	Version history:
	Date        | Version   | Author        | Remark
	----------------------------------------------------------------------------------------
	24/05/2019  | 0.1       | S. Nikodem    | First release MHS TIA 15.1
	14/06/2019  | 0.2       | M. Kurc       | Replacement of instruction if for direct write into variable, temporary variables review
	14/06/2019  | 0.3       | M. Kurc       | Communication error corrected
	19/06/2019  | 0.4       | M. Kurc       | Deleting error word
	25/06/2019  | 0.6       | M. Kurc       | Change interface q_UDT_VFDStatistic to iq_UDT_VFDStatistic
	04/07/2019  | 0.7       | S. Nikodem    | Add auto-parametrization fuction
	18/07/2019  | 0.8       | M. Kurc       | Deleting functions (denormaliztion, normalization, rpm-mm/s, mm/s-rpm)
	24/07/2019  | 2.0       | L. Klar       | 2.0 MHS library release TIA 15.1
	14/08.2019  | 2.1       | K. Pokorski   | Profinet number and HWID reading logic added
	09/09/2019  | 2.2       | S. Nikodem    | Complete rebuild block
	17/09/2019  | 2.3       | S. Nikodem    | Add ramp start/stop
	30/09/2019  | 2.4       | K. Pokorski   | Changed region 1 contents to FC
	30/09/2019  | 2.5       | K. Pokorski   | Implemented new VFD status
	30/09/2019  | 2.6       | L. Klar       | Actual speed connected to a new interface UDT, UDT interface changed
	11/10/2019  | 2.7       | S. Nikodem    | Added Interlock, quick stop, default ramp start/stop time = 20s, running statistic
	30/10/2019  | 2.8       | K. Pokorski   | Acceleration and deceleration calculating fixed
	30/10/2019  | 2.9       | K. Pokorski   | Internal warning and error handling changed
	20/11/2019  | 2.10      | S. Nikodem    | Configuration error
	20/11/2019  | 3.0       | P.Majka       | 3.0 MHS library release TIA 15.1
	03/12/2019  | 3.1       | S. Nikodem    | Change of direction
	20/12/2019  | 3.2       | S. Deulkar    | Used configureation error bit to report to conveyor block
	28/01/2020  | 3.3       | S. Nikodem    | Configuration error if speed setpoint is too high
	06/02/2020  | 3.4       | S. Nikodem    | Configuration error - Simulation mode bypass PNDeviceFound
	02/01/2020  | 3.5       | F.Baten       | Changed "UDT_VFD_Status" to be without positioning status
	04/03/2020  | 3.6       | F.Baten       | Output speed scaling based on measured speed at fixed output value, removal of gearratio and wheelendperrimeter
	01/05/2020  | 3.7       | F.Baten       | Reverted 3.6 modification measured speed
	18/06/2020  | 3.8       | L.Klar        | ix_PowerOK splitted to 24vOK and 400vOK
	23/06/2020  | 3.9       | L.Klar        | VFD running change to cover deceleration ramp, at speed condition changed to have False in standstill
	08/07/2020  | 3.10      | S.Theocharis  | Change VFD acknowledge to extended pulse & send acknowledge even with PN Slave error
	09/07/2020  | 3.11      | S.Theocharis  | Updated PO UDT
	10/07/2020  | 3.12      | S.Theocharis  | Comment out the PNSlave error from the VfdAvailable and ErrorActive variables to allo run in a ring topology
	22/07/2020  | 3.13      | K.Pokorski    | Protection against negative actual speed (int overflow)
	14/09/2020  | 3.14      | S.Nikodem     | VFDRunningFeedback error
	03/11/2020  | 3.15      | K.Pokorski    | Profinet ports diagnostics added
	06/01/2022  | 3.16      | M.Roijen      | Update new FB_Commissioning block
	21/02/2023  | 4.0       | F.Baten       | 4.0 Release TIA 17.5
	    *)

	REGION 1 - Get Device Profinet information

	    "FC_GetDevicePN"(is_PNDeviceName := #iUDT_VfdConfig.VFDPNDeviceName,
	                     ix_SimulationModeActive := #ix_SimulationModeActive,
	                     iqUDT_PND := #sUDT_PNDevice);


	    "FC_GetPNPortStatus"(ii_NumberOfPorts := #ci_NumberOfProfinetPorts,
	                         iUDT_DevicePNInfo := #sUDT_PNDevice,
	                         qa_PortFault => #sa_PNPortsStatus);

	END_REGION

	REGION 2 - Reset errors

	    IF #iqUDT_ConveyorInterface.InternalErrorReset                           // Reser errors when Reset is given
	    THEN

	        #sUDT_Status.PNSlaveNotonline := FALSE;
	        #sUDT_Status.PNSlaveError := FALSE;
	        #sUDT_Status.InternalError := FALSE;
	        #sUDT_Status.VFDRunningFeedbackError := FALSE;
	        #sUDT_Status.PNSlaveWarning := FALSE;

	    END_IF;


	    // Create  extended pulse for VFD Reset
	    #sFB_TimerOnOffDelayVFDReset(iudi_OnDelayTime := 0,
	                                 iudi_OffDelayTime := 200,
	                                 ix_SignalToDelay := #iqUDT_ConveyorInterface.InternalErrorReset,
	                                 ix_Enable := TRUE);

	END_REGION

	REGION 3 - Hardware checks
	    // Hardware will only be available after the delay, so the device has time for the initialisation
	    #sFB_TimerOnOffDelayCheck24V(iudi_OnDelayTime := 2000,
	                                 ix_SignalToDelay := #ix_24vOk);

	    #sx_24vOk := #sFB_TimerOnOffDelayCheck24V.qx_DelayedSignal;

	    #sFB_TimerOnOffDelayCheck400V(iudi_OnDelayTime := 2000,
	                                  ix_SignalToDelay := #ix_400vOk);

	    #sx_400vOk := #sFB_TimerOnOffDelayCheck400V.qx_DelayedSignal;

	    // Check if PN device is online
	    IF NOT "DB_ProfinetDiagnostic".ProfinetNetworks[#sUDT_PNDevice.PNNetworknumber].DeviceStatus[#sUDT_PNDevice.PNDeviceNumber].DeviceState.Exist
	        AND NOT #ix_SimulationModeActive
	        AND #sx_24vOk
	    THEN
	        #sUDT_Status.PNSlaveNotonline := TRUE;

	    END_IF;

	    // Check if PN ports are healthy
	    IF #sa_PNPortsStatus[1] XOR #sa_PNPortsStatus[2] THEN
	        #sUDT_Status.PNSlaveWarning := TRUE;
	    END_IF;


	    // Check if PN device has an error
	    IF "DB_ProfinetDiagnostic".ProfinetNetworks[#sUDT_PNDevice.PNNetworknumber].DeviceStatus[#sUDT_PNDevice.PNDeviceNumber].DeviceState.Error
	        AND NOT #ix_SimulationModeActive
	        AND #sx_24vOk
	        AND NOT #sUDT_Status.PNSlaveWarning
	    THEN
	        #sUDT_Status.PNSlaveError := TRUE;
	    END_IF;

	    // Set bit when PN device is healthy (online and no error)
	    #sx_PNDeviceHealthy := NOT #sUDT_Status.PNSlaveNotonline
	    AND NOT #sUDT_Status.PNSlaveError
	    AND #sUDT_PNDevice.PNDeviceFound
	    AND #sx_24vOk;

	    // Set hardware available bit when all conditions are met
	    #sx_HardwareAvailable := (#sx_24vOk
	    AND #sx_PNDeviceHealthy)
	    OR #ix_SimulationModeActive;


	    // VFD is ready for operation if hardware ok
	    #sx_VFD_Available := #sx_HardwareAvailable;

	END_REGION

	REGION 4 - Check errors and warnings

	    // Check if the VFD has a warning
	    #sUDT_Status.InternalWarning := #iUDT_VfdInputs.ZSW_1.AlarmActive;

	    // Copy warning code to status DB when warning active
	    IF #iUDT_VfdInputs.ZSW_1.AlarmActive
	    THEN

	        #sUDT_Status.ErrorCode := UINT_TO_INT(#iUDT_VfdInputs.AlarmCode);

	    END_IF;

	    // Check if the VFD has an error
	    #sUDT_Status.InternalError := #iUDT_VfdInputs.ZSW_1.FaultActive AND NOT #sx_StartMeasuring;

	    // Copy error code to status DB when error active
	    IF #iUDT_VfdInputs.ZSW_1.FaultActive
	    THEN

	        #sUDT_Status.ErrorCode := UINT_TO_INT(#iUDT_VfdInputs.FaultCode);

	    END_IF;

	    // Reset error code if warning and error not available
	    IF (NOT #iUDT_VfdInputs.ZSW_1.AlarmActive
	        AND NOT #iUDT_VfdInputs.ZSW_1.FaultActive)
	    THEN

	        #sUDT_Status.ErrorCode := 0;

	    END_IF;

	END_REGION

	REGION 5 - Check if configuration is ok for commissioning purposes

	    IF #iUDT_VfdConfig.WheelEndPerimeter > 0.0                                         // If perimeter of wheel at the end of gear is greater than 0
	        AND #iUDT_VfdConfig.GearRatio > 0.0                                            // and gear ratio is greater than 0
	        AND #iUDT_VfdConfig.ReferenceRPM > 0.0                                             // and maximum speed is greater than 0
	        AND #iUDT_VfdConfig.VFDRampUpTime > 0                                          // and ramp up time is greater than 0
	        AND #iUDT_VfdConfig.VFDRampDownTime > 0                                        // and ramp down time is greater than zero
	        AND #iUDT_VfdConfig.VFDStartupTime > 0.0                                       // and startup time is greater then zero
	        AND 2 * #cudi_DefaultRampUpTime > #iUDT_VfdConfig.VFDRampUpTime                // and ramp up time is not greater two time than default ramp up time
	        AND 2 * #cudi_DefaultRampDownTime > #iUDT_VfdConfig.VFDRampDownTime            // and ramp down time is not greater two time than default ramp down time

	        AND (#sUDT_PNDevice.PNDeviceFound                                              // and device not found in PN structure
	        OR #ix_SimulationModeActive)                                                    // or simulation mode is active
	    THEN
	        #sx_ConfigurationError := FALSE;                                                // Reset configuration error
	    ELSE
	        #sx_ConfigurationError := TRUE;                                                 // Set configuration error
	    END_IF;

	END_REGION

	REGION 6 - Speed handling

	    // Calculate actual speed in mm/s
	    #si_ActualSpeed := REAL_TO_INT((((INT_TO_REAL(#iUDT_VfdInputs.ActualSpeed) / #cr_MaximumOutput) * #iUDT_VfdConfig.ReferenceRPM) / #iUDT_VfdConfig.GearRatio) * #iUDT_VfdConfig.WheelEndPerimeter / 60.0);

	    // Reversal actual speed
	    IF #iUDT_VfdConfig.DirectionReversal THEN

	        #si_ActualSpeed := #si_ActualSpeed * -1;

	    END_IF;

	    // Calculate actual speed setpoint
	    #sr_ActualSpeedSetpoint := ((DINT_TO_REAL(INT_TO_DINT(#iqUDT_ConveyorInterface.SpeedSetpoint) * 60) / #iUDT_VfdConfig.WheelEndPerimeter) * #iUDT_VfdConfig.GearRatio);

	    // Check if speed setpoint is reached
	    #sx_SpeedSetpointReached := (ABS(#si_ActualSpeed) >= (#iqUDT_ConveyorInterface.SpeedSetpoint - #iUDT_VfdConfig.SpeedSetpointWindow))
	    AND (ABS(#si_ActualSpeed) <= (#iqUDT_ConveyorInterface.SpeedSetpoint + #iUDT_VfdConfig.SpeedSetpointWindow));
	END_REGION

	REGION 7 - Prepare output data VFD
	    REGION 7.1 - Set speed setpoint in forward and reverse directory

	        // If motor stopped and Run forward is requested and interlock forward is active, the speed setpoint is loaded to run forward.
	        IF (#iUDT_VfdInputs.ActualSpeed = 0) AND #iqUDT_ConveyorInterface.RunFwd AND #iUDT_VfdConfig.InterlockFwd
	        THEN
	            #sx_RunVFDForward := TRUE;
	            #sx_RunVFDReverse := FALSE;
	        END_IF;

	        // If motor stopped and Run reverse is requested and interlock reverse is active, the speed setpoint is loaded to run reverse.
	        IF (#iUDT_VfdInputs.ActualSpeed = 0) AND #iqUDT_ConveyorInterface.RunRvs AND #iUDT_VfdConfig.InterlockRvs
	        THEN
	            #sx_RunVFDReverse := TRUE;
	            #sx_RunVFDForward := FALSE;
	        END_IF;

	    END_REGION

	    REGION 7.2 - Stopping

	        // Create trigger when direction signal falling
	        #sF_TRIG_RunFwd(CLK := #iqUDT_ConveyorInterface.RunFwd);
	        #sF_TRIG_RunRvs(CLK := #iqUDT_ConveyorInterface.RunRvs);

	        // When no run signal is given the VFD should stop
	        IF NOT #iqUDT_ConveyorInterface.RunRvs AND NOT #iqUDT_ConveyorInterface.RunFwd
	            OR (#iqUDT_ConveyorInterface.RunRvs AND #iqUDT_ConveyorInterface.RunFwd)
	            OR #sF_TRIG_RunRvs.Q
	            OR #sF_TRIG_RunFwd.Q

	        THEN
	            #sx_RunVFDReverse := FALSE;
	            #sx_RunVFDForward := FALSE;
	        END_IF;

	        IF NOT #sx_RunVFDReverse AND NOT #sx_RunVFDForward AND (#iUDT_VfdInputs.ActualSpeed <> 0)
	        THEN
	            #sx_VFDStopping := TRUE;
	        ELSE
	            #sx_VFDStopping := FALSE;
	        END_IF;

	    END_REGION

	    REGION 7.3 - Check for enable operation signal

	        #sx_EnableOperation := #sx_VFD_Available AND #sx_400vOk AND NOT #sx_ConfigurationError AND (#sx_RunVFDForward OR #sx_RunVFDReverse); // add communication error

	    END_REGION

	    REGION 7.4 - Write acceleration and deceleration value to drive
	        // Write accceleration value to VFD
	        #qUDT_VfdOutputs.SetpointAcceleration := REAL_TO_INT(#cr_MaximumOutput / UDINT_TO_REAL(#cudi_DefaultRampUpTime) * UDINT_TO_REAL(#iUDT_VfdConfig.VFDRampUpTime));        //Recalculating Acceleration ramp

	        // Write deceleration value to VFD
	        #qUDT_VfdOutputs.SetpointDeceleration := REAL_TO_INT(#cr_MaximumOutput / UDINT_TO_REAL(#cudi_DefaultRampDownTime) * UDINT_TO_REAL(#iUDT_VfdConfig.VFDRampDownTime));      //Recalculating Deceleration ramp

	    END_REGION

	END_REGION

	REGION 8 - Auto Commisioning

	    REGION 8.1 Extract telegram's HW_ID

	        IF (#ix_StartCommissioning)
	        THEN

	            #si_Log2GeoReturn := LOG2GEO(LADDR := "DB_ProfinetDiagnostic".ProfinetNetworks[#sUDT_PNDevice.PNNetworknumber].DeviceStatus[#sUDT_PNDevice.PNDeviceNumber].DeviceState.HW_ID, GEOADDR := #sv_VFDGeoStruct);       // "LOG2GEO" to get profinet network number
	            #sv_VFDGeoStruct.AREA := #ci_VFDArea;                                                                                                                                                                               // Set IO Profinet devices area ID
	            #sv_VFDGeoStruct.HWTYPE := #ci_SubmoduleHWType;                                                                                                                                                                     // Set submodule HW_type number
	            #sv_VFDGeoStruct.STATION := INT_TO_UINT(#sUDT_PNDevice.PNDeviceNumber);                                                                                                                                            // Set device's profinet number
	            #sv_VFDGeoStruct.SLOT := #ci_TelegramSlot;                                                                                                                                                                          // Set free telegram slot
	            #sv_VFDGeoStruct.SUBSLOT := #ci_TelegramSubslot;                                                                                                                                                                    // Set free telegram subslot

	            #si_Geo2LogReturn := GEO2LOG(GEOADDR := #sv_VFDGeoStruct, LADDR => #shw_VFD_Telegram);                                                                                                                              // "GEO2LOG" to get free telegram's HW_ID

	        END_IF;

	    END_REGION

	    REGION 8.2 Run auto - commissioning

	        // Using commissioning block to write/read parameter. Start parametrization if rise edge trigger from start commissionig signal
	        #sFB_Commissioning(ix_Enable := #ix_StartCommissioning,
	                           ihw_SinaParamHardwareId := #shw_VFD_Telegram,                    // Set hardware id ,
	                           iUDT_MotorConfig := #iUDT_MotorData,
	                           qx_StartMeasuring => #sx_StartMeasuring,                         // Set start measuring signal
	                           iqx_GoToNextStep := #iqx_GoToNextStepCommissioning);             // Set/Reset signal go to next step


	    END_REGION ;

	END_REGION

	REGION 9 - Write outputs to VFD

	    REGION 9.1 - Write control word 1


	        #qUDT_VfdOutputs.STW_1.ControlViaPLC := TRUE;
	        #qUDT_VfdOutputs.STW_1.DirectionReversal := FALSE;
	        #qUDT_VfdOutputs.STW_1.ONOFF1 := #sx_EnableOperation OR #sx_StartMeasuring;
	        #qUDT_VfdOutputs.STW_1.OFF2 := TRUE;
	        #qUDT_VfdOutputs.STW_1.OFF3 := #ix_QuickStopDisable;
	        #qUDT_VfdOutputs.STW_1.EnableOperation := #sx_RunVFDReverse OR #sx_RunVFDForward OR #iUDT_VfdInputs.ActualSpeed <> 0 OR #sx_StartMeasuring;
	        #qUDT_VfdOutputs.STW_1.DoNotDisableRFG := TRUE;
	        #qUDT_VfdOutputs.STW_1.EnableRFG := TRUE;
	        #qUDT_VfdOutputs.STW_1.EnableSetpoint := TRUE;
	        #qUDT_VfdOutputs.STW_1.Acknowledge := #sFB_TimerOnOffDelayVFDReset.qx_DelayedSignal;


	        IF (NOT #sx_VFD_Available OR NOT #sx_400vOk) AND NOT #sx_StartMeasuring
	        THEN

	            #qUDT_VfdOutputs.STW_1.ForceDormantErrorTest := FALSE;
	            #qUDT_VfdOutputs.STW_1.SpareBit9 := FALSE;
	            #qUDT_VfdOutputs.STW_1.DirectionReversal := FALSE;
	            #qUDT_VfdOutputs.STW_1.SpareBit12 := FALSE;
	            #qUDT_VfdOutputs.STW_1.SpareBit13 := FALSE;
	            #qUDT_VfdOutputs.STW_1.SpareBit14 := FALSE;
	            #qUDT_VfdOutputs.STW_1.SpareBit15 := FALSE;
	            #qUDT_VfdOutputs.STW_1.ONOFF1 := FALSE;
	            #qUDT_VfdOutputs.STW_1.OFF2 := FALSE;
	            #qUDT_VfdOutputs.STW_1.OFF3 := FALSE;
	            #qUDT_VfdOutputs.STW_1.EnableOperation := FALSE;
	            #qUDT_VfdOutputs.STW_1.DoNotDisableRFG := FALSE;
	            #qUDT_VfdOutputs.STW_1.EnableRFG := FALSE;
	            #qUDT_VfdOutputs.STW_1.EnableSetpoint := FALSE;
	            #qUDT_VfdOutputs.SpeedSetpoint := 0;

	        END_IF;

	    END_REGION

	    REGION 9.2 - Write speed setpoint to drive

	        // Calculate normalized speed setpoint
	        #qUDT_VfdOutputs.SpeedSetpoint := REAL_TO_INT((#sr_ActualSpeedSetpoint / #iUDT_VfdConfig.ReferenceRPM) * #cr_MaximumOutput);
	        IF #qUDT_VfdOutputs.SpeedSetpoint > #cr_MaximumOutput
	        THEN
	            #qUDT_VfdOutputs.SpeedSetpoint := REAL_TO_INT(#cr_MaximumOutput);
	        END_IF;

	        // The conveyor stopped and may now run in reverse direction
	        IF (#sx_RunVFDReverse AND NOT #iUDT_VfdConfig.DirectionReversal)
	            OR (#sx_RunVFDForward AND #iUDT_VfdConfig.DirectionReversal)
	        THEN
	            #qUDT_VfdOutputs.SpeedSetpoint := #qUDT_VfdOutputs.SpeedSetpoint * -1;
	        END_IF;

	        // Clear speed setpoint when no run request or above direction request or is configuration error
	        IF (NOT #sx_RunVFDForward AND NOT #sx_RunVFDReverse)
	            OR #sx_ConfigurationError
	        THEN
	            #qUDT_VfdOutputs.SpeedSetpoint := 0;
	        END_IF;

	    END_REGION

	END_REGION

	REGION 10 - Check if motor is running

	    //The moto should start running after specific time. If not the VFDRunningFeedback error occured
	    #sFB_TimerOnOffDelayVFDRunningFeedbackError(iudi_OnDelayTime := #iUDT_VfdConfig.VFDStartupTime,
	                                                ix_SignalToDelay := #sx_EnableOperation AND NOT (#si_ActualSpeed <> 0));

	    IF #sFB_TimerOnOffDelayVFDRunningFeedbackError.qx_DelayedSignal THEN

	        #sUDT_Status.VFDRunningFeedbackError := TRUE;

	    END_IF;

	END_REGION

	REGION 11 - Copy signals to interface DB and to status output UDT
	    // Create internal error status
	    #sx_ErrorActive := #sUDT_Status.PNSlaveNotonline
	    OR #sUDT_Status.VFDRunningFeedbackError
	    //  OR #s_UDT_Status.PNSlaveError Commented out by AST to allow run in ring topology v3.12
	    OR #sUDT_Status.InternalError;

	    // Write interface bits
	    #iqUDT_ConveyorInterface.VFDRunning := #iUDT_VfdInputs.ZSW_1.Ready AND #sx_VFD_Available AND (#iqUDT_ConveyorInterface.ActualSpeed <> 0 OR #iUDT_VfdInputs.ZSW_1.OperationEnabled);   // Write true on output Conveyor interface structure if VFD is in operation and motor is turning
	    #iqUDT_ConveyorInterface.VFDatSpeed := #sx_SpeedSetpointReached AND #sx_VFD_Available AND #si_ActualSpeed <> 0;                                                                                                  // Copy setpoint speed reached state from static to the output conveyor interface structure
	    #iqUDT_ConveyorInterface.InternalWarningVFD := #iUDT_VfdInputs.ZSW_1.AlarmActive;                                                                                                      // Set the internal VFD warning bit if any warning is active
	    #iqUDT_ConveyorInterface.InternalErrorVFD := #sx_ErrorActive;                                                                                                                           // Set the internal VFD error bit if any fault is active
	    #iqUDT_ConveyorInterface.ActualSpeed := #si_ActualSpeed;                                                                                                                                // Copy the calculated value to the output
	    #iqUDT_ConveyorInterface.ConfigurationError := #iqUDT_ConveyorInterface.ConfigurationError OR #sx_ConfigurationError;

	    // Copy error status to output
	    #qUDT_HMIStatus := #sUDT_Status;

	END_REGION

	REGION 12 - Statistic
	    // Create trigger on error and create statistics for profinet slave not online
	    #sR_TRIG_PNSlaveNotOnline(CLK := #sUDT_Status.PNSlaveNotonline);                                        // Detect the rising edge of the error

	    IF #iqUDT_ConveyorInterface.ResetStatistics OR #sUDT_Status.PNSlaveNotonline
	    THEN

	        "FC_Statistics"(ix_Reset := #iqUDT_ConveyorInterface.ResetStatistics,
	                        ix_Activate := #sUDT_Status.PNSlaveNotonline,
	                        ix_RTrigActivate := #sR_TRIG_PNSlaveNotOnline.Q,
	                        iqUDT_Statistics := #iqUDT_VfdStatistics.PNSlaveNotOnline);
	    END_IF;

	    // Create trigger on error and create statistics for profinet slave error
	    #sR_TRIG_PNSlaveError(CLK := #sUDT_Status.PNSlaveError);                                        // Detect the rising edge of the error

	    IF #iqUDT_ConveyorInterface.ResetStatistics OR #sUDT_Status.PNSlaveError
	    THEN

	        "FC_Statistics"(ix_Reset := #iqUDT_ConveyorInterface.ResetStatistics,
	                        ix_Activate := #sUDT_Status.PNSlaveError,
	                        ix_RTrigActivate := #sR_TRIG_PNSlaveError.Q,
	                        iqUDT_Statistics := #iqUDT_VfdStatistics.PNSlaveError);
	    END_IF;

	    // Create trigger on error and create statistics for internal VFD Error
	    #sR_TRIG_VFDInternalError(CLK := #sUDT_Status.InternalError);                                        // Detect the rising edge of the error

	    IF #iqUDT_ConveyorInterface.ResetStatistics OR #sUDT_Status.InternalError
	    THEN

	        "FC_Statistics"(ix_Reset := #iqUDT_ConveyorInterface.ResetStatistics,
	                        ix_Activate := #sUDT_Status.InternalError,
	                        ix_RTrigActivate := #sR_TRIG_VFDInternalError.Q,
	                        iqUDT_Statistics := #iqUDT_VfdStatistics.VFDInternalError);
	    END_IF;

	    // Create trigger on running signal and create statistics for running status
	    #sR_TRIG_Running(CLK := #iqUDT_ConveyorInterface.VFDRunning);                                        // Detect the rising edge of the signal

	    IF #iqUDT_ConveyorInterface.ResetStatistics OR #iqUDT_ConveyorInterface.VFDRunning
	    THEN

	        "FC_Statistics"(ix_Reset := #iqUDT_ConveyorInterface.ResetStatistics,
	                        ix_Activate := #iqUDT_ConveyorInterface.VFDRunning,
	                        ix_RTrigActivate := #sR_TRIG_Running.Q,
	                        iqUDT_Statistics := #iqUDT_VfdStatistics.Running);
	    END_IF;

	END_REGION
END_FUNCTION_BLOCK

FUNCTION_BLOCK "FB_Unloader"
TITLE = FB_Unloader
{ S7_Optimized_Access := 'TRUE' }
AUTHOR : MHSE
FAMILY : Equimpent
VERSION : 3.0
// ATTRIBUTES
// AUTO_NUMBER = True
// BLOCK_NUMBER = 232
// END_ATTRIBUTES
//Function block to control unloader.
   VAR_INPUT
      iUDT_UnloaderConfiguration { ExternalAccessible := 'False'; ExternalVisible := 'False'; ExternalWritable := 'False'} : "UDT_UnloaderConfiguration";   //   Unloader configuration structure
      ix_SafetyReset { ExternalAccessible := 'False'; ExternalVisible := 'False'; ExternalWritable := 'False'} : Bool;   //  Safety reset
      ix_SafetyOk { ExternalAccessible := 'False'; ExternalVisible := 'False'; ExternalWritable := 'False'} : Bool;   //   TRUE when Safety Circuit of the Conveyor is healthy
      ix_24vOk { ExternalAccessible := 'False'; ExternalVisible := 'False'; ExternalWritable := 'False'} : Bool;   //   TRUE when 24VDC is healthy
      ix_400vOk { ExternalAccessible := 'False'; ExternalVisible := 'False'; ExternalWritable := 'False'} : Bool;   //   TRUE when 400VAC is healthy
      ix_ProfinetOk { ExternalAccessible := 'False'; ExternalVisible := 'False'; ExternalWritable := 'False'} : Bool;   //   TRUE when the PN node(s) of VSU are OK
      ix_ReadyUnload { ExternalAccessible := 'False'; ExternalVisible := 'False'; ExternalWritable := 'False'} : Bool;   //   TRUE when Unloader is ready to unload
      ix_Running { ExternalAccessible := 'False'; ExternalVisible := 'False'; ExternalWritable := 'False'} : Bool;   //   TRUE when Unloader is running
      ix_TooLongParcel { ExternalAccessible := 'False'; ExternalVisible := 'False'; ExternalWritable := 'False'} : Bool;   //   TRUE when Unloader has detected a too long parcel (stopped)
      ix_VFDError { ExternalAccessible := 'False'; ExternalVisible := 'False'; ExternalWritable := 'False'} : Bool;   //   TRUE when Unloader has an VFD error
      ix_Healthy { ExternalAccessible := 'False'; ExternalVisible := 'False'; ExternalWritable := 'False'} : Bool;   //   TRUE when Unloader has no Errors
      ix_PECEoS { ExternalAccessible := 'False'; ExternalVisible := 'False'; ExternalWritable := 'False'} : Bool;   //   TRUE when the end of section photoeye is not blocked
      ix_ManualControlled { ExternalAccessible := 'False'; ExternalVisible := 'False'; ExternalWritable := 'False'} : Bool;   //   Unloader is controlled by
      ix_ExternalRequestDieBack { ExternalAccessible := 'False'; ExternalVisible := 'False'; ExternalWritable := 'False'} : Bool;   //   External request die back
      ix_ExternalRequestHold { ExternalAccessible := 'False'; ExternalVisible := 'False'; ExternalWritable := 'False'} : Bool;   //   External request hold
      ix_ResetEnergySave { ExternalAccessible := 'False'; ExternalVisible := 'False'; ExternalWritable := 'False'} : Bool;   //   Reset energy save mode timer
      ix_HardwareOk { ExternalAccessible := 'False'; ExternalVisible := 'False'; ExternalWritable := 'False'} : Bool;   //  TRUE when  hardware is Ok
   END_VAR

   VAR_OUTPUT
      qUDT_HMIStatus { ExternalAccessible := 'False'; ExternalVisible := 'False'; ExternalWritable := 'False'} : "UDT_UnloaderStatus";   //   HMI status structure
      qUDT_Status { ExternalAccessible := 'False'; ExternalVisible := 'False'; ExternalWritable := 'False'} : "UDT_CommonStatus";   //   Common status structure
      qi_SpeedSelect { ExternalAccessible := 'False'; ExternalVisible := 'False'; ExternalWritable := 'False'} : Int;   //   Speed select (slow, normal or fast)
      qx_ReleaseUnload { ExternalAccessible := 'False'; ExternalVisible := 'False'; ExternalWritable := 'False'} : Bool;   //   Release Unloader
      qx_EStopReset { ExternalAccessible := 'False'; ExternalVisible := 'False'; ExternalWritable := 'False'} : Bool;
      qx_FaultReset { ExternalAccessible := 'False'; ExternalVisible := 'False'; ExternalWritable := 'False'} : Bool;
   END_VAR

   VAR_IN_OUT
      iqUDT_EquipmentControl : "UDT_EquipmentControl";   //   Equipment control structure
      iqUDT_UnloaderCommand : "UDT_UnloaderCommand";   //   Unloader HMI control
      iqUDT_HandShake : "UDT_ConveyorHandshake";   //   Handshake structure
      iqUDT_EquipmentInterface : "UDT_ConveyorInterface";   //   Equipment interface structure
      iqUDT_Statistics : "UDT_UnloaderStatistics";   //   Statistics structure
   END_VAR

   VAR
      sUDT_CommonStatus { ExternalAccessible := 'False'; ExternalVisible := 'False'; ExternalWritable := 'False'; S7_SetPoint := 'False'} : "UDT_CommonStatus";   //   Common status structure
      sUDT_CommonStatusOld { ExternalAccessible := 'False'; ExternalVisible := 'False'; ExternalWritable := 'False'; S7_SetPoint := 'False'} : "UDT_CommonStatus";   //   Auxiliary status structure
      sUDT_HMIStatus { ExternalAccessible := 'False'; ExternalVisible := 'False'; ExternalWritable := 'False'; S7_SetPoint := 'False'} : "UDT_UnloaderStatus";   //   HMI status structure
      s_FB_TimerOnOffDelaySafetyOKPulse { ExternalAccessible := 'False'; ExternalVisible := 'False'; ExternalWritable := 'False'; S7_SetPoint := 'False'} : "FB_TimerOnOffDelay";
      sFB_PECEoSFiltered { ExternalAccessible := 'False'; ExternalVisible := 'False'; ExternalWritable := 'False'; S7_SetPoint := 'False'} : "FB_TimerOnOffDelay";   //   Filtering end of section photo eye signal
      sFB_PECEoSJamTimer { ExternalAccessible := 'False'; ExternalVisible := 'False'; ExternalWritable := 'False'; S7_SetPoint := 'False'} : "FB_TimerOnOffDelay";   //   Timer to detect photo eye jam
      sFB_EnergySaveTimer { ExternalAccessible := 'False'; ExternalVisible := 'False'; ExternalWritable := 'False'; S7_SetPoint := 'False'} : "FB_TimerOnOffDelay";   //   Timer to start energy save mode
      sFB_PEC { ExternalAccessible := 'False'; ExternalVisible := 'False'; ExternalWritable := 'False'; S7_SetPoint := 'False'} : "FB_PEC";   //   FB PEC block for PEC Jam status
      sR_TRIG_PEC_EoSFiltered {InstructionName := 'R_TRIG'; LibVersion := '1.0'; ExternalAccessible := 'False'; ExternalVisible := 'False'; ExternalWritable := 'False'; S7_SetPoint := 'False'} : R_TRIG;   //   Rising edge trigger end of section photo eye filtered
      sF_TRIG_PEC_EoSFiltered {InstructionName := 'F_TRIG'; LibVersion := '1.0'; ExternalAccessible := 'False'; ExternalVisible := 'False'; ExternalWritable := 'False'; S7_SetPoint := 'False'} : F_TRIG;   //   Falling edge trigger end of section photo eye filtered
      sR_TRIG_EnergySave {InstructionName := 'R_TRIG'; LibVersion := '1.0'; ExternalAccessible := 'False'; ExternalVisible := 'False'; ExternalWritable := 'False'; S7_SetPoint := 'False'} : R_TRIG;   //   Rising edge for energy save
      sR_TRIG_ConveyorUp {InstructionName := 'R_TRIG'; LibVersion := '1.0'; ExternalAccessible := 'False'; ExternalVisible := 'False'; ExternalWritable := 'False'; S7_SetPoint := 'False'} : R_TRIG;   //   Rising edge of automatic active
      sR_TRIG_ConveyorDown {InstructionName := 'R_TRIG'; LibVersion := '1.0'; ExternalAccessible := 'False'; ExternalVisible := 'False'; ExternalWritable := 'False'; S7_SetPoint := 'False'} : R_TRIG;   //   Rising edge of automatic not active
      sR_TRIG_VFDError {InstructionName := 'R_TRIG'; LibVersion := '1.0'; ExternalAccessible := 'False'; ExternalVisible := 'False'; ExternalWritable := 'False'; S7_SetPoint := 'False'} : R_TRIG;   //   Rising edge of VFD error
      sR_TRIG_NotHealthy {InstructionName := 'R_TRIG'; LibVersion := '1.0'; ExternalAccessible := 'False'; ExternalVisible := 'False'; ExternalWritable := 'False'; S7_SetPoint := 'False'} : R_TRIG;   //   Rising edge trigger if extendable not healthy
      sR_TRIG_TooLongParcel {InstructionName := 'R_TRIG'; LibVersion := '1.0'; ExternalAccessible := 'False'; ExternalVisible := 'False'; ExternalWritable := 'False'; S7_SetPoint := 'False'} : R_TRIG;   //   Rising edge trigger for too long parcel
      s_R_TRIG_SafetyOK {InstructionName := 'R_TRIG'; LibVersion := '1.0'; ExternalAccessible := 'False'; ExternalVisible := 'False'; ExternalWritable := 'False'; S7_SetPoint := 'False'} : R_TRIG;
      si_AuxEnergySave { ExternalAccessible := 'False'; ExternalVisible := 'False'; ExternalWritable := 'False'} : Int;   //   Auxiliery energy save
      sx_Disabled { ExternalAccessible := 'False'; ExternalVisible := 'False'; ExternalWritable := 'False'} : Bool;   //   Operation is enabled
      sx_Ready { ExternalAccessible := 'False'; ExternalVisible := 'False'; ExternalWritable := 'False'} : Bool;   //   Conveyor Ready to operate in Automatic mode
      sx_StartReceived { ExternalAccessible := 'False'; ExternalVisible := 'False'; ExternalWritable := 'False'} : Bool;   //   Start command received from system
      sx_PEC_EoSFiltered { ExternalAccessible := 'False'; ExternalVisible := 'False'; ExternalWritable := 'False'} : Bool;   //   End of section photo eye filtered
      sx_EnergySaveActive { ExternalAccessible := 'False'; ExternalVisible := 'False'; ExternalWritable := 'False'} : Bool;   //   Active energy save mode
      sx_AutomaticActive { ExternalAccessible := 'False'; ExternalVisible := 'False'; ExternalWritable := 'False'} : Bool;   //   Automatic active
   END_VAR


BEGIN
	(*
	----------------------------------------------------------------------------------------

	Version history:
	Date        | Version   | Author        | Remark
	----------------------------------------------------------------------------------------
	24/05/2019  | 0.1       | F.Baten       | first release MHS TIA 15.1
	17/06/2019  | 0.3       | L.Klar        | Manual mode added to "UDT_EquipmentControl"
	24/07/2019  | 2.0       | L.Klar        | 2.0 MHS library release TIA 15.1
	14/10/2019  | 2.1       | L.Klar        | Updated status structure
	15/10/2019  | 2.2       | S.Deulkar     | Deleted unused symbol, added statistcs, rearrange structure
	04/11/2019  | 2.3       | L.Klar        | First scan bit changed from memory bit to DB variable
	12/11/2019  | 3.0       | P.Majka       | 3.0 MHS library release TIA 15.1
	04/03/2020  | 3.1       | P.Majka       | Adapting reviews, repair statistics for too long parcels
	31/03/2020  | 3.2       | F.Baten       | UDT_UnloaderCommand added
	                                        | Disable by HMI added
	22/09/2020  | 3.3       | L.Klar        | Reset added
	11/01/2021  | 3.4       | L.Klar        | Input safety ok added to stop conveyor condition
	27/02/2021  | 3.5       | M. Kurpiers   | Button disable/enable operation and status fixed
	02/03/2021  | 3.6       | K. Pokorski   | Halted and dieback status enable only when automatic on
	13/03/2021  | 3.7       | L.Klar        | HMI status updated- warning commented, energy save added
	13/03/2021  | 3.8       | L.Klar        | Energy save corrected
	08/04/2021  | 3.9       | K.Pokorski    | VFD error masked when safety is not ok
	21/02/2023  | 4.0       | F.Baten       | 4.0 Release TIA 17.5
	*)

	REGION 1 - Initial

	    REGION 1.1 - First PLC cycle

	        // Bits initialization.
	        IF "DB_Memory".FirstScan
	        THEN
	            #qx_ReleaseUnload := FALSE;
	            #sx_AutomaticActive := FALSE;
	            #sx_StartReceived := FALSE;
	            #sx_Disabled := FALSE;
	        END_IF;

	    END_REGION

	    REGION 1.2 Triggers

	        // Rising edge trigger end of section photo eye filtered.
	        #sR_TRIG_PEC_EoSFiltered(CLK := #sx_PEC_EoSFiltered);

	        // Falling edge trigger end of section photo eye filtered.
	        #sF_TRIG_PEC_EoSFiltered(CLK := #sx_PEC_EoSFiltered);

	        // Rising edge trigger energy save.
	        #sR_TRIG_EnergySave(CLK := #sUDT_CommonStatus.EnergySave);

	        // Rising edge extendable up.
	        #sR_TRIG_ConveyorUp(CLK := #sx_AutomaticActive AND #sx_Ready);

	        // Rising edge extendable down.
	        #sR_TRIG_ConveyorDown(CLK := #sx_AutomaticActive AND NOT #sx_Ready);

	        // Rising edge extendable VFD error.
	        #sR_TRIG_VFDError(CLK := #sUDT_HMIStatus.Specific.VFDError);

	        // Rising edge extendable not healthy.
	        #sR_TRIG_NotHealthy(CLK := #sUDT_HMIStatus.Specific.NotHealthy);

	        // Rising edge for too long parcel.
	        #sR_TRIG_TooLongParcel(CLK := #sUDT_HMIStatus.Specific.TooLongParcel);

	    END_REGION

	    REGION HMI button Disable/Enable operation
	        IF #iqUDT_UnloaderCommand.Disable
	        THEN
	            #sx_Disabled := TRUE;
	        ELSE
	            #sx_Disabled := FALSE;
	        END_IF;

	        #iqUDT_UnloaderCommand.Disable := FALSE;


	        // Copy status to HMI
	        #sUDT_HMIStatus.Specific.Disabled := #sx_Disabled;

	    END_REGION

	END_REGION

	REGION 2 - Errors

	    // PEC EoS.
	    #sFB_PEC(ix_PEC := #ix_PECEoS,
	             iUDT_PECConfiguration := #iUDT_UnloaderConfiguration.PEC_EOS,
	             qx_PECFiltered => #sx_PEC_EoSFiltered,
	             qUDT_HMIStatus => #sUDT_HMIStatus.Specific.PEC_EoS,
	             iqUDT_ConveyorInterface := #iqUDT_EquipmentInterface,
	             iqUDT_PECStatistics := #iqUDT_Statistics.PEC_EOS);

	    // Parcel too long.
	    #sUDT_HMIStatus.Specific.TooLongParcel := #ix_TooLongParcel;

	    // VFD Error.
	    #sUDT_HMIStatus.Specific.VFDError := (#ix_VFDError AND #ix_400vOk AND #ix_ProfinetOk AND #ix_SafetyOk);

	    // Not healthy.
	    #sUDT_HMIStatus.Specific.NotHealthy := (NOT #ix_Healthy AND #ix_400vOk AND #ix_24vOk AND #ix_ProfinetOk);

	    // Common Error.
	    #sUDT_CommonStatus.Error := NOT #ix_24vOk
	    OR NOT #ix_400vOk
	    OR NOT #ix_ProfinetOk
	    OR NOT #ix_SafetyOk
	    OR #sUDT_HMIStatus.Specific.PEC_EoS.Jam
	    OR #sUDT_HMIStatus.Specific.VFDError
	    OR #sUDT_HMIStatus.Specific.NotHealthy;

	    // Warning.
	    #sUDT_CommonStatus.Warning := #sUDT_HMIStatus.Specific.TooLongParcel;

	END_REGION

	REGION 3 - Check conditions to set unloader ready

	    // Ready to operate.
	    #sx_Ready := NOT #sUDT_CommonStatus.Error
	    AND #ix_Healthy
	    AND NOT #ix_ManualControlled;

	END_REGION

	REGION 4 - Stop unloader

	    // Reset bits to stop unloader.
	    IF NOT #iqUDT_EquipmentControl.Command.AutomaticOn
	        OR #sUDT_CommonStatus.Error
	        OR NOT #ix_Healthy
	        OR #ix_ManualControlled
	        OR NOT #ix_SafetyOk
	    THEN
	        #qx_ReleaseUnload := FALSE;
	        #sx_AutomaticActive := FALSE;
	        #sx_StartReceived := FALSE;
	    END_IF;

	END_REGION

	REGION 5 - Start Automatic mode

	    // If start (one shot) is received from system, this is memorised until started in cascade.
	    IF #iqUDT_EquipmentControl.Command.Start
	        AND #sx_Ready
	    THEN
	        #sx_StartReceived := TRUE;
	    END_IF;

	    // Activating automatic mode.
	    IF #sx_StartReceived
	        AND (#iqUDT_HandShake.CascadeStartUp
	        OR #iUDT_UnloaderConfiguration.FirstConveyorToStart)
	    THEN
	        #sx_AutomaticActive := TRUE;
	        #sx_StartReceived := FALSE;
	    END_IF;

	END_REGION

	REGION 6 - Automatic mode active

	    REGION 6.1 - Ready To Send (RTS)

	        // Set Ready to send signal.
	        IF #sF_TRIG_PEC_EoSFiltered.Q
	            AND #sx_AutomaticActive
	            AND #sx_Ready
	            AND #ix_ReadyUnload
	        THEN
	            #iqUDT_HandShake.RTS := TRUE;
	        END_IF;

	        // Reset Ready to send signal.
	        IF #sR_TRIG_PEC_EoSFiltered.Q
	        THEN
	            #iqUDT_HandShake.RTS := FALSE;
	        END_IF;

	    END_REGION

	    REGION 6.2 - Operation

	        // Run Unloader.
	        #qx_ReleaseUnload := #sx_AutomaticActive
	        AND #sx_Ready
	        AND #ix_ReadyUnload
	        AND ((#iqUDT_HandShake.RTR
	        AND NOT #ix_ExternalRequestDieBack)
	        OR #sx_PEC_EoSFiltered)
	        AND NOT #sx_Disabled
	        AND NOT #ix_ExternalRequestHold
	        AND NOT #sx_EnergySaveActive;

	    END_REGION

	    REGION 6.3 - Energy save

	        IF #iUDT_UnloaderConfiguration.Energy THEN

	            // Set Energy save active.
	            IF #si_AuxEnergySave >= #iUDT_UnloaderConfiguration.EnergySaveLength
	            THEN
	                #sx_EnergySaveActive := TRUE;
	            END_IF;

	            // Reset or increment displacement calculation to use for energy save.
	            IF NOT #sx_PEC_EoSFiltered
	                OR #ix_ResetEnergySave
	                OR #ix_ManualControlled
	                //OR NOT #ix_ReadyUnload
	            THEN
	                #si_AuxEnergySave := 0;
	                #sx_EnergySaveActive := FALSE;
	            ELSE
	                #si_AuxEnergySave += #iqUDT_EquipmentInterface.Displacement;
	            END_IF;

	        ELSE

	            #si_AuxEnergySave := 0;
	            #sx_EnergySaveActive := FALSE;

	        END_IF;

	    END_REGION

	END_REGION

	REGION 7 - Speed control

	    // Copy speed setpoint from configuration.
	    #qi_SpeedSelect := #iUDT_UnloaderConfiguration.Speedsetpoint;

	    // Clear speed setpoint depending on wrong configuration.
	    IF #iUDT_UnloaderConfiguration.Speedsetpoint < 0
	        OR #iUDT_UnloaderConfiguration.Speedsetpoint > 2
	    THEN
	        #qi_SpeedSelect := 0;
	    END_IF;

	END_REGION

	REGION 8 - Reset

	    // Safety ok extended pulse
	    #s_R_TRIG_SafetyOK(CLK := #ix_SafetyReset);

	    #s_FB_TimerOnOffDelaySafetyOKPulse(iudi_OffDelayTime := 1000,
	                                       ix_SignalToDelay := #s_R_TRIG_SafetyOK.Q);

	    // Fault and Estop reset outputs
	    #qx_FaultReset := #ix_SafetyReset OR #iqUDT_EquipmentControl.Command.Reset OR #s_FB_TimerOnOffDelaySafetyOKPulse.qx_DelayedSignal;
	    #qx_EStopReset := #ix_SafetyReset OR #s_FB_TimerOnOffDelaySafetyOKPulse.qx_DelayedSignal;

	END_REGION

	REGION 9 - Statistics

	    // Up time.
	    IF #sx_AutomaticActive
	        AND #sx_Ready
	        OR #iqUDT_EquipmentControl.Command.ResetData
	    THEN
	        "FC_Statistics"(ix_Reset := #iqUDT_EquipmentControl.Command.ResetData,
	                        ix_Activate := #sx_AutomaticActive AND #sx_Ready,
	                        ix_RTrigActivate := #sR_TRIG_ConveyorUp.Q,
	                        iqUDT_Statistics := #iqUDT_Statistics.ExtendableUpTime);
	    END_IF;

	    // Down time.
	    IF #sx_AutomaticActive
	        AND #sx_Ready
	        OR #iqUDT_EquipmentControl.Command.ResetData
	    THEN
	        "FC_Statistics"(ix_Reset := #iqUDT_EquipmentControl.Command.ResetData,
	                        ix_Activate := #sx_AutomaticActive AND NOT #sx_Ready,
	                        ix_RTrigActivate := #sR_TRIG_ConveyorDown.Q,
	                        iqUDT_Statistics := #iqUDT_Statistics.ExtendableDownTime);
	    END_IF;

	    // Energy save mode active.
	    IF #sx_EnergySaveActive
	        OR #iqUDT_EquipmentControl.Command.ResetData
	    THEN
	        "FC_Statistics"(ix_Reset := #iqUDT_EquipmentControl.Command.ResetData,
	                        ix_Activate := #sUDT_CommonStatus.EnergySave,

	                        ix_RTrigActivate := #sR_TRIG_EnergySave.Q,
	                        iqUDT_Statistics := #iqUDT_Statistics.EnergySave);
	    END_IF;

	    // VFD Error.
	    IF #sUDT_HMIStatus.Specific.VFDError
	        OR #iqUDT_EquipmentControl.Command.ResetData
	    THEN
	        "FC_Statistics"(ix_Reset := #iqUDT_EquipmentControl.Command.ResetData,
	                        ix_Activate := #sUDT_HMIStatus.Specific.VFDError,
	                        ix_RTrigActivate := #sR_TRIG_VFDError.Q,
	                        iqUDT_Statistics := #iqUDT_Statistics.VFDError);
	    END_IF;

	    // Not healthy .
	    IF #sUDT_HMIStatus.Specific.NotHealthy
	        OR #iqUDT_EquipmentControl.Command.ResetData
	    THEN
	        "FC_Statistics"(ix_Reset := #iqUDT_EquipmentControl.Command.ResetData,
	                        ix_Activate := #sUDT_HMIStatus.Specific.NotHealthy,
	                        ix_RTrigActivate := #sR_TRIG_NotHealthy.Q,
	                        iqUDT_Statistics := #iqUDT_Statistics.NotHealthy);
	    END_IF;

	    // Too long parcel.
	    IF #sUDT_HMIStatus.Specific.TooLongParcel
	        OR #iqUDT_EquipmentControl.Command.ResetData
	    THEN
	        "FC_Statistics"(ix_Reset := #iqUDT_EquipmentControl.Command.ResetData,
	                        ix_Activate := #sUDT_HMIStatus.Specific.TooLongParcel,
	                        ix_RTrigActivate := #sR_TRIG_TooLongParcel.Q,
	                        iqUDT_Statistics := #iqUDT_Statistics.TooLongParcel);
	    END_IF;

	END_REGION

	REGION 10 - Status

	    // Set statuses.
	    #sUDT_CommonStatus.Stopped := NOT #sx_AutomaticActive;
	    #sUDT_CommonStatus.Running := #ix_Running;
	    #sUDT_CommonStatus.AutoON := #sx_Ready AND #sx_AutomaticActive;
	    #sUDT_CommonStatus.Halted := #ix_ExternalRequestHold AND #sUDT_CommonStatus.AutoON AND NOT #sx_EnergySaveActive;
	    #sUDT_CommonStatus.Dieback := (NOT #iqUDT_HandShake.RTR OR #ix_ExternalRequestDieBack) AND #sUDT_CommonStatus.AutoON AND NOT #sx_EnergySaveActive
	    AND NOT #sUDT_CommonStatus.EnergySave AND NOT #sUDT_CommonStatus.Running;
	    #sUDT_CommonStatus.Manual := #ix_ManualControlled;
	    #sUDT_CommonStatus.ManualRun := #sUDT_CommonStatus.Manual AND #sUDT_CommonStatus.Running;
	    #sUDT_CommonStatus.EnergySave := #sx_EnergySaveActive;
	    #sUDT_CommonStatus.SafetyStop := NOT #ix_SafetyOk;


	    // HMI status update on change.
	    IF #sUDT_CommonStatusOld <> #sUDT_CommonStatus
	    THEN
	        // HMI status initialization.
	        #sUDT_HMIStatus.Status := 0;

	        // Energy save.
	        IF #sUDT_CommonStatus.EnergySave
	        THEN
	            #sUDT_HMIStatus.Status := "DB_HMIStatusConfiguration".EnergySave;
	        END_IF;

	        // Running.
	        IF #sUDT_CommonStatus.Running
	        THEN
	            #sUDT_HMIStatus.Status := "DB_HMIStatusConfiguration".Running;
	        END_IF;

	        // Stopped.
	        IF #sUDT_CommonStatus.Stopped
	        THEN
	            #sUDT_HMIStatus.Status := "DB_HMIStatusConfiguration".Stopped;
	        END_IF;

	        // Dieback.
	        IF #sUDT_CommonStatus.Dieback
	        THEN
	            #sUDT_HMIStatus.Status := "DB_HMIStatusConfiguration".Dieback;
	        END_IF;

	        // Halted.
	        IF #sUDT_CommonStatus.Halted
	        THEN
	            #sUDT_HMIStatus.Status := "DB_HMIStatusConfiguration".Halted;
	        END_IF;

	        // Dimension error.
	        IF #sUDT_HMIStatus.Specific.TooLongParcel
	        THEN
	            #sUDT_HMIStatus.Status := "DB_HMIStatusConfiguration".DimensionError;
	        END_IF;

	        // Manual.
	        IF #sUDT_CommonStatus.Manual
	        THEN
	            #sUDT_HMIStatus.Status := "DB_HMIStatusConfiguration".Manual;
	        END_IF;

	        // Running in manual mode.
	        IF #sUDT_CommonStatus.ManualRun
	        THEN
	            #sUDT_HMIStatus.Status := "DB_HMIStatusConfiguration".ManualRun;
	        END_IF;

	        //  PEC error.
	        IF #sUDT_HMIStatus.Specific.PEC_EoS.Jam
	        THEN
	            #sUDT_HMIStatus.Status := "DB_HMIStatusConfiguration".PECJam;
	        END_IF;

	        // Not healthy.
	        IF #sUDT_HMIStatus.Specific.NotHealthy
	        THEN
	            #sUDT_HMIStatus.Status := "DB_HMIStatusConfiguration".VFDNotHealthy;
	        END_IF;

	        // VFD error.
	        IF #sUDT_HMIStatus.Specific.VFDError
	        THEN
	            #sUDT_HMIStatus.Status := "DB_HMIStatusConfiguration".VFDError;
	        END_IF;

	        // Safety stop.
	        IF #sUDT_CommonStatus.SafetyStop
	        THEN
	            #sUDT_HMIStatus.Status := "DB_HMIStatusConfiguration".SafetyStop;
	        END_IF;

	        // Copy statuses.

	        #sUDT_CommonStatusOld := #sUDT_CommonStatus;


	    END_IF;

	    #qUDT_HMIStatus := #sUDT_HMIStatus;
	    #qUDT_Status := #sUDT_CommonStatus;

	END_REGION

	REGION 11 - Report to control block

	    "FC_EquipmentReport"(iUDT_Status := #sUDT_CommonStatus,
	                         iqUDT_Control := #iqUDT_EquipmentControl);

	END_REGION
END_FUNCTION_BLOCK

FUNCTION_BLOCK "FB_TCPIPConnect"
TITLE = FB_TCPIPConnect
{ S7_Optimized_Access := 'TRUE' }
AUTHOR : MHSE
FAMILY : Communication
VERSION : 3.0
// ATTRIBUTES
// AUTO_NUMBER = True
// BLOCK_NUMBER = 231
// END_ATTRIBUTES
//Function block to establish and terminateTCPIP connection.
   VAR_INPUT
      iUDT_Connection { ExternalAccessible := 'False'; ExternalVisible := 'False'; ExternalWritable := 'False'} : "UDT_Connection";   // Connection parameters
   END_VAR

   VAR_OUTPUT
      qUDT_HMIStatus { ExternalAccessible := 'False'; ExternalVisible := 'False'; ExternalWritable := 'False'} : "UDT_TCPIPConnectStatus";   // HMI status structure
      qUDT_Status { ExternalAccessible := 'False'; ExternalVisible := 'False'; ExternalWritable := 'False'} : "UDT_CommonStatus";   // Common status structure
      qx_Connected { ExternalAccessible := 'False'; ExternalVisible := 'False'; ExternalWritable := 'False'} : Bool;   // Connected status
   END_VAR

   VAR_IN_OUT
      iqUDT_EquipmentControl : "UDT_EquipmentControl";   // Equipment control structure
      iqUDT_Statistics : "UDT_TCPIPConnectStatistics";   // Statistic structure
      iqx_Reconnect { ExternalAccessible := 'False'; ExternalVisible := 'False'; ExternalWritable := 'False'} : Bool;   // Reconnect command
   END_VAR

   VAR
      sUDT_CommonStatus { ExternalAccessible := 'False'; ExternalVisible := 'False'; ExternalWritable := 'False'; S7_SetPoint := 'False'} : "UDT_CommonStatus";   // Common status structure
      sFB_TCON {InstructionName := 'TCON'; LibVersion := '4.0'; ExternalAccessible := 'False'; ExternalVisible := 'False'; ExternalWritable := 'False'; S7_SetPoint := 'False'} : TCON;   // Siemens "TCON" block - to establish the connection
      sFB_TDISCON {InstructionName := 'TDISCON'; LibVersion := '2.1'; ExternalAccessible := 'False'; ExternalVisible := 'False'; ExternalWritable := 'False'; S7_SetPoint := 'False'} : TDISCON;   // Siemens "TDISCON" block - to terminate the connection
      sFB_DIAG {InstructionName := 'T_DIAG'; LibVersion := '1.2'; ExternalAccessible := 'False'; ExternalVisible := 'False'; ExternalWritable := 'False'; S7_SetPoint := 'False'} : T_DIAG;   // Siemens "T_DIAG" block - to diagnose the connection
      sFB_TimerConTimeout { ExternalAccessible := 'False'; ExternalVisible := 'False'; ExternalWritable := 'False'; S7_SetPoint := 'False'} : "FB_TimerOnOffDelay";   // MHS "FB_TimerOnOffDelay" block - to measure the connection timeout
      sFB_TimerFilter { ExternalAccessible := 'False'; ExternalVisible := 'False'; ExternalWritable := 'False'; S7_SetPoint := 'False'} : "FB_TimerOnOffDelay";   // MHS "FB_TimerOnOffDelay" block - to filter the connection established signal
      sv_InterfaceData {InstructionName := 'TCON_IP_v4'; LibVersion := '1.0'; ExternalAccessible := 'False'; ExternalVisible := 'False'; ExternalWritable := 'False'; S7_SetPoint := 'False'} : TCON_IP_v4;   // TCON Interface configuration data
      sR_TRIG_ConnectionLost {InstructionName := 'R_TRIG'; LibVersion := '1.0'; ExternalAccessible := 'False'; ExternalVisible := 'False'; ExternalWritable := 'False'; S7_SetPoint := 'False'} : R_TRIG;   // Siemens "R_TRIG" - to prepare rising edge signal on Connection lost signal
      sR_TRIG_Reset {InstructionName := 'R_TRIG'; LibVersion := '1.0'; ExternalAccessible := 'False'; ExternalVisible := 'False'; ExternalWritable := 'False'; S7_SetPoint := 'False'} : R_TRIG;   // Siemens "R_TRIG" - to prepare rising edge signal on reset data signal
      sa_Connect { ExternalAccessible := 'False'; ExternalVisible := 'False'; ExternalWritable := 'False'} : Struct   // TCON interface structure
         Request { ExternalAccessible := 'False'; ExternalVisible := 'False'; ExternalWritable := 'False'} : Bool;   //  TCON - Request
         Done { ExternalAccessible := 'False'; ExternalVisible := 'False'; ExternalWritable := 'False'} : Bool;   //  TCON - Done
         Busy { ExternalAccessible := 'False'; ExternalVisible := 'False'; ExternalWritable := 'False'} : Bool;   //  TCON - Busy
         Error { ExternalAccessible := 'False'; ExternalVisible := 'False'; ExternalWritable := 'False'} : Bool;   //  TCON - Error
         Active { ExternalAccessible := 'False'; ExternalVisible := 'False'; ExternalWritable := 'False'} : Bool;   //  TCON - Active
         Status { ExternalAccessible := 'False'; ExternalVisible := 'False'; ExternalWritable := 'False'} : Word;   //  TCON - Status
      END_STRUCT;
      sa_Disconnect { ExternalAccessible := 'False'; ExternalVisible := 'False'; ExternalWritable := 'False'} : Struct   // TDISCON interface structure
         Request { ExternalAccessible := 'False'; ExternalVisible := 'False'; ExternalWritable := 'False'} : Bool;   //  TDISCON - Request
         Done { ExternalAccessible := 'False'; ExternalVisible := 'False'; ExternalWritable := 'False'} : Bool;   //  TDISCON - Done
         Busy { ExternalAccessible := 'False'; ExternalVisible := 'False'; ExternalWritable := 'False'} : Bool;   //  TDISCON - Busy
         Error { ExternalAccessible := 'False'; ExternalVisible := 'False'; ExternalWritable := 'False'} : Bool;   //  TDISCON - Error
         Active { ExternalAccessible := 'False'; ExternalVisible := 'False'; ExternalWritable := 'False'} : Bool;   //  TDISCON - Active
         Status { ExternalAccessible := 'False'; ExternalVisible := 'False'; ExternalWritable := 'False'} : Word;   //  TDISCON - Status
      END_STRUCT;
      sa_Diag { ExternalAccessible := 'False'; ExternalVisible := 'False'; ExternalWritable := 'False'} : Struct   // T_DIAG block diagnostic variables
         Request { ExternalAccessible := 'False'; ExternalVisible := 'False'; ExternalWritable := 'False'} : Bool;   //  TDIAG - Request
         Done { ExternalAccessible := 'False'; ExternalVisible := 'False'; ExternalWritable := 'False'} : Bool;   //  TDIAG - Done
         Busy { ExternalAccessible := 'False'; ExternalVisible := 'False'; ExternalWritable := 'False'} : Bool;   //  TDIAG - Busy
         Error { ExternalAccessible := 'False'; ExternalVisible := 'False'; ExternalWritable := 'False'} : Bool;   //  TDIAG - Error
         Active { ExternalAccessible := 'False'; ExternalVisible := 'False'; ExternalWritable := 'False'} : Bool;   //  TDIAG - Active
         Status { ExternalAccessible := 'False'; ExternalVisible := 'False'; ExternalWritable := 'False'} : Word;   //  TDIAG - Status
         Result {InstructionName := 'TDiag_Status'; LibVersion := '1.0'; ExternalAccessible := 'False'; ExternalVisible := 'False'; ExternalWritable := 'False'} : TDiag_Status;   //  TDIAG - Result
      END_STRUCT;
      sx_Connected { ExternalAccessible := 'False'; ExternalVisible := 'False'; ExternalWritable := 'False'} : Bool;   // Connection established memory
      sx_ConnectedFiltred { ExternalAccessible := 'False'; ExternalVisible := 'False'; ExternalWritable := 'False'} : Bool;   // Connection established memory (filtred)
      sx_CommunicationFault { ExternalAccessible := 'False'; ExternalVisible := 'False'; ExternalWritable := 'False'} : Bool;   // Communication fault
   END_VAR


BEGIN
	(*
	----------------------------------------------------------------------------------------

	Version history:
	Date        | Version   | Author        | Remark
	----------------------------------------------------------------------------------------
	24/05/2019  | 0.1       | L.Klar        | first release MHS TIA 15.1
	13/06/2019  | 0.2       | A.Nowak       | Delete writing to variable - S_FB_Timer_ConTimeout
	24/06/2019  | 0.3       | L.Klar        | Status running added
	25/06/2019  | 0.5       | L.Klar        | Statistics changed to InOut
	24/07/2019  | 2.0       | L.Klar        | 2.0 MHS library release TIA 15.1
	21/08/2019  | 2.1       | K.Pokorski    | Comments adjusted
	26/09/2019  | 2.2       | A.Nowak       | Delete static status structure and change region 9. Create new static sx_CommunicationFault.
	09/10/2019  | 2.3       | M.Kurc        | System equipment control added
	04/11/2019  | 2.4       | L.Klar        | 10 Hz clock and first scan changed from memory bit to DB variable
	19/11/2019  | 2.5       | L.Klar        | Status outputs corrected
	20/11/2019  | 3.0       | P.Majka       | 3.0 MHS library release TIA 15.1
	21/02/2023  | 4.0       | F.Baten       | 4.0 Release TIA 17.5
	*)

	REGION 1 – Initialization

	    // Reset connected status bit and reconnect command bit during first PLC scan
	    IF ("DB_Memory".FirstScan)             // First PLC scan occured
	    THEN

	        #sx_Connected := FALSE;
	        #iqx_Reconnect := TRUE;

	    END_IF;

	END_REGION

	REGION 2 – Connection error reset

	    // Reset errors and blocks statuses when no connection state available and communication fault reset received
	    #sR_TRIG_Reset(CLK := #iqUDT_EquipmentControl.Command.Reset);

	    IF (#sx_CommunicationFault                                      // Communication fault
	        AND #sR_TRIG_Reset.Q)                                      // Reset signal trigger
	    THEN

	        #sa_Connect.Status := 16#0;
	        #sa_Disconnect.Status := 16#0;
	        #sa_Diag.Status := 16#0;
	        #sx_CommunicationFault := FALSE;

	    END_IF;

	END_REGION

	REGION 3 – Communication Interface preparation

	    #sv_InterfaceData.InterfaceId := #iUDT_Connection.Interface_ID;                       // HW-identifier of IE-interface submodule
	    #sv_InterfaceData.ID := #iUDT_Connection.ID;                                          // Connection reference / identifier
	    #sv_InterfaceData.ConnectionType := 16#0B;                                             // Type OF connection: 11=TCP/IP, 19=UDP 17=TCP/IP
	    #sv_InterfaceData.ActiveEstablished := #iUDT_Connection.ActiveEstablished;            // Active/passive connection establishment
	    #sv_InterfaceData.RemoteAddress.ADDR[1] := INT_TO_BYTE(#iUDT_Connection.IP[1]);       // Remote IP address (IPv4) - x.0.0.0
	    #sv_InterfaceData.RemoteAddress.ADDR[2] := INT_TO_BYTE(#iUDT_Connection.IP[2]);       // Remote IP address (IPv4) - 0.x.0.0
	    #sv_InterfaceData.RemoteAddress.ADDR[3] := INT_TO_BYTE(#iUDT_Connection.IP[3]);       // Remote IP address (IPv4) - 0.0.x.0
	    #sv_InterfaceData.RemoteAddress.ADDR[4] := INT_TO_BYTE(#iUDT_Connection.IP[4]);       // Remote IP address (IPv4) - 0.0.0.x

	    // Set local or remote port depending on whether the PLC is active or passive device in connection
	    IF (#sv_InterfaceData.ActiveEstablished)                                               // Active connection
	    THEN

	        #sv_InterfaceData.LocalPort := 0;
	        #sv_InterfaceData.RemotePort := #iUDT_Connection."Port";

	        // Passive connection
	    ELSE

	        #sv_InterfaceData.LocalPort := #iUDT_Connection."Port";
	        #sv_InterfaceData.RemotePort := 0;

	    END_IF;

	END_REGION

	REGION 4 – Connection establishment and termination

	    IF (#iqx_Reconnect)                                                     // Reconnect request
	    THEN

	        // Terminate a TCPIP connection if reconnect command available and connection established
	        IF (#sx_Connected)                                                  // Connection established
	        THEN

	            // Disconnect request
	            #sa_Disconnect.Request :=
	            #iqx_Reconnect                                                  // Reconnect command
	            AND #sa_Disconnect.Status = 16#7000;                            // TDISCON block status is equal to 16#7000 (No job processing active)

	            // Terminate a TCPIP connection when request available
	            #sFB_TDISCON(REQ := #sa_Disconnect.Request,
	                         ID := #sv_InterfaceData.ID,
	                         DONE => #sa_Disconnect.Done,
	                         BUSY => #sa_Disconnect.Busy,
	                         ERROR => #sa_Disconnect.Error,
	                         STATUS => #sa_Disconnect.Status);

	            // In case of connection broken, connected bit and disconnect block active bit are reset
	            IF (#sa_Disconnect.Done)                                        // Disconnect was successful
	            THEN

	                #sx_Connected := FALSE;
	                #sa_Disconnect.Active := FALSE;

	                // Connection termination in progress
	            ELSE

	                #sa_Disconnect.Active := TRUE;                              // Set the disconnecting active status bit

	            END_IF;

	            // Try to establish connection if reconnect command active and there is no connection
	        ELSE                                                                // Connection is terminated

	            // Connect request
	            #sa_Connect.Request := #iqx_Reconnect AND                       // Reconnect command
	            #sa_Connect.Status = 16#7000;            // TCON block status is equal to 16#7000 (No job processing active)

	            // Establishing a TCPIP connection when request available
	            #sFB_TCON(REQ := #sa_Connect.Request,
	                      ID := #sv_InterfaceData.ID,
	                      DONE => #sa_Connect.Done,
	                      BUSY => #sa_Connect.Busy,
	                      ERROR => #sa_Connect.Error,
	                      STATUS => #sa_Connect.Status,
	                      CONNECT := #sv_InterfaceData);

	            // In case of connection established, connected bit is set, connect block active bit and reconnect command are reset
	            IF (#sa_Connect.Done)                                           // Connect successful
	            THEN

	                #sx_Connected := TRUE;
	                #sa_Connect.Active := FALSE;
	                #iqx_Reconnect := FALSE;

	                // Connection establishing in progress
	            ELSE

	                #sa_Connect.Active := TRUE;                                 // Set the connecting active status

	            END_IF;

	        END_IF;

	    END_IF;

	END_REGION

	REGION 5 – Connection establishment and termination error handling

	    // Measure the maximum connect or disconnect time
	    #sFB_TimerConTimeout(ix_SignalToDelay := #sa_Connect.Active
	                         OR #sa_Disconnect.Active,
	                         iudi_OnDelayTime := DINT_TO_UDINT(#iUDT_Connection.ConTimeout),
	                         iudi_OffDelayTime := 0);

	    IF (#sFB_TimerConTimeout.qx_DelayedSignal)                                                 // Connecting / disconnecting time error from connection timeout timer
	    THEN

	        IF (#sa_Connect.Active)                                                                  // Connecting is active
	        THEN

	            // If connection already exist and block try establish connection, connected bit is set, connect block active bit and reconnect command are reset
	            IF (#sa_Connect.Status = 16#80A3)                                                    // Connecting status equal to 16#80A3 - The connection already exist
	            THEN

	                #sx_Connected := TRUE;
	                #sa_Connect.Active := FALSE;
	                #iqx_Reconnect := FALSE;

	                // Connection time has expired - error generated
	            ELSE

	                #sx_CommunicationFault := TRUE;

	            END_IF;

	            // Disconnect operation failed - error generated
	        ELSIF (#sa_Disconnect.Active)
	        THEN

	            #sx_CommunicationFault := TRUE;

	        END_IF;

	    END_IF;

	    // The connection terminated by partner - error generated, connected bit reset and reconnect command request set
	    IF (#sa_Diag.Result.State <> 16#04)                         // The connection terminated by partner
	    THEN

	        #sx_CommunicationFault := TRUE;
	        #sx_Connected := FALSE;
	        #iqx_Reconnect := TRUE;

	    END_IF;

	END_REGION

	REGION 6 – Connection diagnostic

	    // Check connection condition ten times per second
	    IF (NOT #sa_Connect.Active AND NOT #sa_Disconnect.Active)        // Connecting and disconnecting procedure are not active
	    THEN

	        #sFB_DIAG(REQ := "DB_Memory".Clock_10Hz,
	                  ID := #sv_InterfaceData.ID,
	                  DONE => #sa_Diag.Done,
	                  BUSY => #sa_Diag.Busy,
	                  ERROR => #sa_Diag.Error,
	                  STATUS => #sa_Diag.Status,
	                  RESULT := #sa_Diag.Result);

	    END_IF;

	END_REGION

	REGION 7 – Connection established filter

	    // Connected status bit filtering
	    #sFB_TimerFilter(ix_SignalToDelay := #sx_Connected,
	                     iudi_OnDelayTime := 50,
	                     qx_DelayedSignal => #sx_ConnectedFiltred);

	END_REGION

	REGION 8 – Statistics

	    // Prepare rising edge of connected status signal
	    #sR_TRIG_ConnectionLost(CLK := NOT #sx_ConnectedFiltred);

	    // Conditions to call "FC_Statistics"
	    IF (NOT #sx_ConnectedFiltred                                                        // No connection
	        OR #iqUDT_EquipmentControl.Command.ResetData)                                  // Reset data
	    THEN

	        "FC_Statistics"(ix_Reset := #iqUDT_EquipmentControl.Command.ResetData,
	                        ix_Activate := NOT #sx_ConnectedFiltred,
	                        ix_RTrigActivate := #sR_TRIG_ConnectionLost.Q,
	                        iqUDT_Statistics := #iqUDT_Statistics.ConnectionLost);

	    END_IF;

	END_REGION

	REGION 9 – Status

	    #sUDT_CommonStatus.Error := #sx_CommunicationFault;                        // Error

	    #sUDT_CommonStatus.AutoON := #sx_ConnectedFiltred;                         // Auto ON

	    #qUDT_HMIStatus.Specific.CommunicationFault := #sx_CommunicationFault;     // Communication faults

	    #qUDT_HMIStatus.Specific.Connected := #sx_ConnectedFiltred;                // Connected

	    IF #sUDT_CommonStatus.AutoON                                               // Auto ON
	    THEN

	        #qUDT_HMIStatus.Status := "DB_HMIStatusConfiguration".AutoON;

	    END_IF;

	    IF #sUDT_CommonStatus.Error                                                // Error
	    THEN

	        #qUDT_HMIStatus.Status := "DB_HMIStatusConfiguration".Error;

	    END_IF;

	END_REGION

	REGION 10 Report to control block

	    // Function to manage report between control block and conveyor block

	    "FC_EquipmentReport"(iUDT_Status := #sUDT_CommonStatus,
	                         iqUDT_Control := #iqUDT_EquipmentControl);

	END_REGION

	REGION 11 – Write outputs

	    #qx_Connected := #sx_Connected;

	END_REGION
END_FUNCTION_BLOCK

FUNCTION_BLOCK "FB_SystemControl"
TITLE = FB_SystemControl
{ S7_Optimized_Access := 'TRUE' }
AUTHOR : MHSE
FAMILY : GeneralSystemFunctions
VERSION : 3.0
// ATTRIBUTES
// AUTO_NUMBER = True
// BLOCK_NUMBER = 230
// END_ATTRIBUTES
//Function block to control the system.
   VAR_INPUT
      iudi_SignalingTime { ExternalAccessible := 'False'; ExternalVisible := 'False'; ExternalWritable := 'False'} : UDInt;   // Signaling time [ms]
      ix_SignalingIOModuleOK { ExternalAccessible := 'False'; ExternalVisible := 'False'; ExternalWritable := 'False'} : Bool;   // Beeper and lamp IO module ok
      ix_HMIConnectionOK { ExternalAccessible := 'False'; ExternalVisible := 'False'; ExternalWritable := 'False'} : Bool;   // TRUE = HMI connection is active
      ix_ExternalError { ExternalAccessible := 'False'; ExternalVisible := 'False'; ExternalWritable := 'False'} : Bool;   // TRUE - External error occurred
      ix_SafetyOK { ExternalAccessible := 'False'; ExternalVisible := 'False'; ExternalWritable := 'False'} : Bool;   // TRUE - Safety OK
      ix_Start { ExternalAccessible := 'False'; ExternalVisible := 'False'; ExternalWritable := 'False'} : Bool;   // Start command from control panel
      ix_Stop { ExternalAccessible := 'False'; ExternalVisible := 'False'; ExternalWritable := 'False'} : Bool;   // Stop command from control panel
      ix_Reset { ExternalAccessible := 'False'; ExternalVisible := 'False'; ExternalWritable := 'False'} : Bool;   // Reset command from control panel
   END_VAR

   VAR_OUTPUT
      qUDT_HMIStatus { ExternalAccessible := 'False'; ExternalVisible := 'False'; ExternalWritable := 'False'} : "UDT_SystemControlStatus";   // HMI status structure
      qUDT_Status { ExternalAccessible := 'False'; ExternalVisible := 'False'; ExternalWritable := 'False'} : "UDT_CommonStatus";   // Status structure
      qx_StartingFlashLamp { ExternalAccessible := 'False'; ExternalVisible := 'False'; ExternalWritable := 'False'} : Bool;   // Flash lamp
      qx_StartingBeeper { ExternalAccessible := 'False'; ExternalVisible := 'False'; ExternalWritable := 'False'} : Bool;   // Beeper starting
      qx_ErrorLamp { ExternalAccessible := 'False'; ExternalVisible := 'False'; ExternalWritable := 'False'} : Bool;   // Equipment error lamp
      qx_SafetyStopLamp { ExternalAccessible := 'False'; ExternalVisible := 'False'; ExternalWritable := 'False'} : Bool;   // Safety stop lamp
      qx_StoppedLamp { ExternalAccessible := 'False'; ExternalVisible := 'False'; ExternalWritable := 'False'} : Bool;   // Equipment stopped lamp
      qx_StartedLamp { ExternalAccessible := 'False'; ExternalVisible := 'False'; ExternalWritable := 'False'} : Bool;   // Equipment started lamp
      qx_WarningLamp { ExternalAccessible := 'False'; ExternalVisible := 'False'; ExternalWritable := 'False'} : Bool;   // Equipment warning lamp
   END_VAR

   VAR_IN_OUT
      iqUDT_SystemControlCommand : "UDT_SystemControlCommand";   // HMI system control structure
      iqUDT_Equipment : "UDT_EquipmentControl";   // Equipment control structure
      iqUDT_Statistics : "UDT_SystemControlStatistics";   // Statistics structure
   END_VAR

   VAR
      sUDT_CommonStatus { ExternalAccessible := 'False'; ExternalVisible := 'False'; ExternalWritable := 'False'; S7_SetPoint := 'False'} : "UDT_CommonStatus";   // Status structure
      sUDT_HMIStatus { ExternalAccessible := 'False'; ExternalVisible := 'False'; ExternalWritable := 'False'; S7_SetPoint := 'False'} : "UDT_SystemControlStatus";   // Status structure
      sUDT_CommonStatusOld { ExternalAccessible := 'False'; ExternalVisible := 'False'; ExternalWritable := 'False'; S7_SetPoint := 'False'} : "UDT_CommonStatus";   // Old status structure
      sUDT_SystemControlCommand { ExternalAccessible := 'False'; ExternalVisible := 'False'; ExternalWritable := 'False'; S7_SetPoint := 'False'} : "UDT_SystemControlCommand";   // HMI system control structure
      sFB_TimerOnOffDelaySignaling { ExternalAccessible := 'False'; ExternalVisible := 'False'; ExternalWritable := 'False'; S7_SetPoint := 'False'} : "FB_TimerOnOffDelay";   // Timer to calculate the signaling time
      sR_TRIG_PB_Start {InstructionName := 'R_TRIG'; LibVersion := '1.0'; ExternalAccessible := 'False'; ExternalVisible := 'False'; ExternalWritable := 'False'; S7_SetPoint := 'False'} : R_TRIG;   // Rising edge for start push button
      sR_TRIG_PB_Stop {InstructionName := 'R_TRIG'; LibVersion := '1.0'; ExternalAccessible := 'False'; ExternalVisible := 'False'; ExternalWritable := 'False'; S7_SetPoint := 'False'} : R_TRIG;   // Rising edge for stop push button
      sR_TRIG_PB_Reset {InstructionName := 'R_TRIG'; LibVersion := '1.0'; ExternalAccessible := 'False'; ExternalVisible := 'False'; ExternalWritable := 'False'; S7_SetPoint := 'False'} : R_TRIG;   // Rising edge for reset push button
      sR_TRIG_SystemStarted {InstructionName := 'R_TRIG'; LibVersion := '1.0'; ExternalAccessible := 'False'; ExternalVisible := 'False'; ExternalWritable := 'False'; S7_SetPoint := 'False'} : R_TRIG;   // Rising edge for system started statistics
      sR_TRIG_SystemError {InstructionName := 'R_TRIG'; LibVersion := '1.0'; ExternalAccessible := 'False'; ExternalVisible := 'False'; ExternalWritable := 'False'; S7_SetPoint := 'False'} : R_TRIG;   // Rising edge for system error statistics
      sR_TRIG_EnergySave {InstructionName := 'R_TRIG'; LibVersion := '1.0'; ExternalAccessible := 'False'; ExternalVisible := 'False'; ExternalWritable := 'False'; S7_SetPoint := 'False'} : R_TRIG;   // Rising edge for system in energy save mode statistics
      sx_SignalingDone { ExternalAccessible := 'False'; ExternalVisible := 'False'; ExternalWritable := 'False'} : Bool;   // Signaling finished
      sx_StartSignalingRequired { ExternalAccessible := 'False'; ExternalVisible := 'False'; ExternalWritable := 'False'} : Bool;   // Start signaling required
      sx_SystemStartup { ExternalAccessible := 'False'; ExternalVisible := 'False'; ExternalWritable := 'False'} : Bool;   // System startup procedure in progress
   END_VAR


BEGIN
	(*
	----------------------------------------------------------------------------------------

	Version history:
	Date        | Version   | Author        | Remark
	----------------------------------------------------------------------------------------
	24/05/2019  | 0.1       | K.Pokorski    | first release MHS TIA 15.1
	17/06/2019  | 0.2       | K.Pokorski    | implementation a new concept
	18/06/2019  | 0.3       | K.Pokorski    | remove reset safety handling
	24/07/2019  | 2.0       | L.Klar        | 2.0 MHS library release TIA 15.1
	28/08/2019  | 2.1       | K.Pokorski    | Correction of block logic and adjusting comments
	13/09/2019  | 2.2       | K.Pokorski    | Lamp outputs added
	14/10/2019  | 2.3       | L.Klar        | Updated status structure
	28/10/2019  | 2.4       | K. Pokorski   | Updated region 1, 6 & 9 - compliance with the new status
	04/11/2019  | 2.5       | L.Klar        | 1 Hz clock and first scan changed from memory bit to DB variable
	20/11/2019  | 2.6       | S. Deulkar    | Always Reseting commads to equipment at the beginning of the block
	21/11/2019  | 3.0       | P.Majka       | 3.0 MHS library release TIA 15.1
	22/05/2020  | 3.1       | M.Roijen      | Disable Start in Signaling handling when in System-Manualmode.
	09/07/2020  | 3.2       | S.Theocharis  | Bug fix in status update. Initialize static status instead output status
	31/07/2020  | 3.3       | S.Theocharis  | Add one shot detection of the push buttons
	11/01/2021  | 3.4       | L.Klar        | iq_UDT_Equipment.Report.SafetyStop removed from automatic on/off
	21/02/2023  | 4.0       | F.Baten       | 4.0 Release TIA 17.5
	12/03/2024  | 4.1       | S. Nieswiec   | Variable name changes according to standard
	*)

	REGION 1 - Push button triggers

	    #sR_TRIG_PB_Start(CLK := #ix_Start);                                            //Start button


	    #sR_TRIG_PB_Stop(CLK := #ix_Stop);                                              //Stop button


	    #sR_TRIG_PB_Reset(CLK := #ix_Reset);                                            //Reset button

	END_REGION


	REGION 2 – HMI and control panel commands handling

	    // Reset all HMI commands during first PLC cycle
	    IF "DB_Memory".FirstScan                                                        // First PLC cycle occurred
	    THEN
	        #iqUDT_SystemControlCommand.Start := FALSE;
	        #iqUDT_SystemControlCommand.Stop := FALSE;
	        #iqUDT_SystemControlCommand.Reset := FALSE;
	        #iqUDT_SystemControlCommand.ResetSafety := FALSE;
	        #iqUDT_SystemControlCommand.ResetData := FALSE;
	        #iqUDT_SystemControlCommand.ManualMode := FALSE;
	        #iqUDT_Equipment.Command.AutomaticOn := FALSE;
	        #iqUDT_Equipment.Command.ManualMode := FALSE;
	        #iqUDT_Equipment.Command.DisableManualMode := FALSE;
	        #iqUDT_Equipment.Request.RestartRequired := FALSE;
	        #iqUDT_Equipment.Request.SignalingRequest := FALSE;
	    END_IF;

	    // Clear commands to equipments
	    #iqUDT_Equipment.Command.Start := FALSE;
	    #iqUDT_Equipment.Command.Stop := FALSE;
	    #iqUDT_Equipment.Command.Reset := FALSE;
	    #iqUDT_Equipment.Command.ResetData := FALSE;

	    // Move HMI control structure to static buffer
	    #sUDT_SystemControlCommand := #iqUDT_SystemControlCommand;

	    // Extension of HMI commands with a commands from control panel
	    #sUDT_SystemControlCommand.Start := #sUDT_SystemControlCommand.Start OR #sR_TRIG_PB_Start.Q;        // Extension of HMI start command with a start command from control panel
	    #sUDT_SystemControlCommand.Stop := #sUDT_SystemControlCommand.Stop OR #sR_TRIG_PB_Stop.Q;           // Extension of HMI stop command with a stop command from control panel
	    #sUDT_SystemControlCommand.Reset := #sUDT_SystemControlCommand.Reset OR #sR_TRIG_PB_Reset.Q;        // Extension of HMI reset command with a reset command from control panel

	END_REGION

	REGION 3 – Signaling handling

	    // Starting signaling time
	    IF ((NOT #ix_ExternalError                                                      // External error not occurred
	        AND (#sUDT_SystemControlCommand.Start                                       // Start command received
	        AND NOT #sUDT_SystemControlCommand.ManualMode                               // Not in manual Mode
	        )
	        AND NOT #sUDT_SystemControlCommand.Stop                                     // Stop command not received
	        AND (#iqUDT_Equipment.Report.Stopped                                        // System stopped
	        OR #iqUDT_Equipment.Request.RestartRequired                                 // Restart Required
	        ))
	        OR #iqUDT_Equipment.Request.SignalingRequest
	        )                                                                           // Equipment request signaling
	        AND #ix_SignalingIOModuleOK                                                 // Signaling module OK

	    THEN

	        #sx_StartSignalingRequired := TRUE;

	        IF (#sUDT_SystemControlCommand.Start)
	        THEN
	            #sx_SystemStartup := TRUE;                                              // Set the system startup flag
	        END_IF;

	        // Stopping signaling time
	    ELSIF (#sUDT_SystemControlCommand.Stop                                          // Stop command from HMI available
	        OR #ix_ExternalError                                                        // Exernal error occured
	        OR NOT #ix_SignalingIOModuleOK)                                             // Signaling module ok
	    THEN
	        #sx_StartSignalingRequired := FALSE;
	        #sx_SystemStartup := FALSE;
	    END_IF;

	    // Measure the signaling time
	    #sFB_TimerOnOffDelaySignaling(iudi_OnDelayTime := #iudi_SignalingTime,
	                                  iudi_OffDelayTime := 0,
	                                  ix_SignalToDelay := #sx_StartSignalingRequired,
	                                  ix_Enable := TRUE,
	                                  qx_DelayedSignal => #sx_SignalingDone);

	END_REGION

	REGION 4 – Automatic ON / OFF

	    // Signaling time elapsed
	    IF (#sx_SignalingDone) THEN

	        #iqUDT_Equipment.Request.SignalingRequest := FALSE;                         // Reset signaling request

	        IF #sx_SystemStartup
	            AND #ix_SafetyOK
	        THEN
	            #iqUDT_Equipment.Command.Start := TRUE;                                 // Start system
	            #iqUDT_Equipment.Command.AutomaticOn := TRUE;                           // And turn on automatic mode
	            #sx_SystemStartup := FALSE;
	        END_IF;

	        IF #sx_SystemStartup
	            OR #ix_SafetyOK
	        THEN
	            #sx_SystemStartup := FALSE;
	        END_IF;

	        #sx_StartSignalingRequired := FALSE;                                        // Reset signaling timer
	        #sx_SignalingDone := FALSE;
	    END_IF;

	    // Stopping system and reset automatic mode command
	    IF #ix_ExternalError                                                            // External error occured
	        OR #sUDT_SystemControlCommand.Stop                                          // Stop command received from HMI
	        OR #sUDT_SystemControlCommand.ManualMode                                    // Manual mode active
	        OR NOT #ix_SafetyOK

	    THEN
	        #iqUDT_Equipment.Command.Stop := TRUE;
	        #iqUDT_Equipment.Command.AutomaticOn := FALSE;
	    END_IF;

	END_REGION

	REGION 5 – Commands to equipment

	    #iqUDT_Equipment.Command.Reset := #sUDT_SystemControlCommand.Reset;             // Move reset HMI command to reset equipment command
	    #iqUDT_Equipment.Command.ResetData := #sUDT_SystemControlCommand.ResetData;     // Move reset data HMI command to reset data equipment command
	    #iqUDT_Equipment.Command.ManualMode := #sUDT_SystemControlCommand.ManualMode;   // Move manual mode HMI command to manual mode equipment command
	    #iqUDT_Equipment.Command.DisableManualMode := NOT #ix_HMIConnectionOK;          // Disable manual mode if HMI connection is broken

	END_REGION

	REGION 6 – Lamp state updating

	    // Light warning before equipment starting. Flashes with a frequency of one period per second.
	    #qx_StartingFlashLamp :=
	    #sx_StartSignalingRequired
	    AND NOT #sx_SignalingDone
	    AND "DB_Memory".Clock_1Hz;

	    // Audiable warning before equipment starting. Intermittent signaling with a frequency of one period per second.
	    #qx_StartingBeeper :=
	    #sx_StartSignalingRequired
	    AND NOT #sx_SignalingDone
	    AND "DB_Memory".Clock_1Hz;

	    // Lamp lighting when an external error or equipment's error occurred
	    #qx_ErrorLamp :=
	    #iqUDT_Equipment.Report.Error
	    OR #ix_ExternalError;

	    // Lamp lighting when the safety error occurred or equipment report the safety stop
	    #qx_SafetyStopLamp :=
	    #iqUDT_Equipment.Report.SafetyStop
	    OR NOT #ix_SafetyOK;

	    // Lamp lighting when the system is stopped
	    #qx_StoppedLamp := NOT #iqUDT_Equipment.Command.AutomaticOn;

	    // Lamp lighting when the system is started
	    #qx_StartedLamp := #iqUDT_Equipment.Report.Running;

	    // Lamp lighting when the equipment report a warning
	    #qx_WarningLamp := #iqUDT_Equipment.Report.Warning;

	END_REGION

	REGION 7 – Equipment state update

	    #sUDT_CommonStatus.EnergySave := #iqUDT_Equipment.Report.EnergySave;                         // Move equipment state "EnergySave" from the equipment structure to status structure
	    #sUDT_CommonStatus.Error := #iqUDT_Equipment.Report.Error;                                   // Move equipment state "Error" from the equipment structure to status structure
	    #sUDT_CommonStatus.Running := #iqUDT_Equipment.Report.Running;                               // Move equipment state "Started" from the equipment structure  to status structure
	    #sUDT_CommonStatus.SafetyStop := #iqUDT_Equipment.Report.SafetyStop OR NOT #ix_SafetyOK;     // Move equipment state "Safety" from the input and the equipment structure to status structure
	    #sUDT_CommonStatus.Stopped := #iqUDT_Equipment.Report.Stopped;                               // Move equipment state "Stopped" from the equipment structure to status structure
	    #sUDT_CommonStatus.Warning := #iqUDT_Equipment.Report.Warning;                               // Move equipment state "Warning" from the equipment structure to status structure
	    #sUDT_CommonStatus.Manual := #iqUDT_Equipment.Report.Manual;                                 // Move equipment state "ManualMode" from the equipment structure to status structure

	END_REGION

	REGION 8 – Status update

	    IF #sUDT_CommonStatus <> #sUDT_CommonStatusOld                                  // Actual status is different than the old one
	    THEN

	        // HMI status initialization
	        #sUDT_HMIStatus.Status := 0;

	        // HMI status calculation
	        IF #sUDT_CommonStatus.EnergySave                                            // Energy save
	        THEN
	            #sUDT_HMIStatus.Status := "DB_HMIStatusConfiguration".EnergySave;
	        END_IF;

	        IF #sUDT_CommonStatus.Running                                               // Running
	        THEN
	            #sUDT_HMIStatus.Status := "DB_HMIStatusConfiguration".Running;
	        END_IF;

	        IF #sUDT_CommonStatus.Stopped                                               // Stopped
	        THEN
	            #sUDT_HMIStatus.Status := "DB_HMIStatusConfiguration".Stopped;
	        END_IF;

	        IF #sUDT_CommonStatus.Dieback                                               // Dieback
	        THEN
	            #sUDT_HMIStatus.Status := "DB_HMIStatusConfiguration".Dieback;
	        END_IF;

	        IF #sUDT_CommonStatus.Halted                                                // Halted
	        THEN
	            #sUDT_HMIStatus.Status := "DB_HMIStatusConfiguration".Halted;
	        END_IF;

	        IF #sUDT_CommonStatus.Manual                                                // Manual
	        THEN
	            #sUDT_HMIStatus.Status := "DB_HMIStatusConfiguration".Manual;
	        END_IF;

	        IF #sUDT_CommonStatus.ManualRun                                             // Running in manual mode
	        THEN
	            #sUDT_HMIStatus.Status := "DB_HMIStatusConfiguration".ManualRun;
	        END_IF;

	        IF #sUDT_CommonStatus.Warning                                               // Warning
	        THEN
	            #sUDT_HMIStatus.Status := "DB_HMIStatusConfiguration".Warning;
	        END_IF;

	        IF #sUDT_CommonStatus.Error                                                 // Error
	        THEN
	            #sUDT_HMIStatus.Status := "DB_HMIStatusConfiguration".Error;
	        END_IF;


	        IF (#sUDT_CommonStatus.SafetyStop)                                          // Safety stop
	        THEN
	            #sUDT_HMIStatus.Status := "DB_HMIStatusConfiguration".SafetyStop;
	        END_IF;


	        #sUDT_CommonStatusOld := #sUDT_CommonStatus;                                // Copy status to memory
	        #qUDT_Status := #sUDT_CommonStatus;

	    END_IF;

	    #qUDT_HMIStatus := #sUDT_HMIStatus;                                            // Copy status to output

	END_REGION

	REGION 9 – Statistics

	    // System started
	    #sR_TRIG_SystemStarted(CLK := #iqUDT_Equipment.Report.Running);                 // The system has started

	    IF #iqUDT_Equipment.Report.Running OR #iqUDT_SystemControlCommand.ResetData     // System running statistics handling
	    THEN
	        "FC_Statistics"(ix_Reset := #iqUDT_SystemControlCommand.ResetData,
	                        ix_Activate := #iqUDT_Equipment.Report.Running,
	                        ix_RTrigActivate := #sR_TRIG_SystemStarted.Q,
	                        iqUDT_Statistics := #iqUDT_Statistics.Run);
	    END_IF;

	    // System error
	    #sR_TRIG_SystemError(CLK := #iqUDT_Equipment.Report.Error);                     // System error occured

	    IF #iqUDT_Equipment.Report.Error OR #iqUDT_SystemControlCommand.ResetData       // Error statistics
	    THEN
	        "FC_Statistics"(ix_Reset := #iqUDT_SystemControlCommand.ResetData,
	                        ix_Activate := #iqUDT_Equipment.Report.Error,
	                        ix_RTrigActivate := #sR_TRIG_SystemError.Q,
	                        iqUDT_Statistics := #iqUDT_Statistics.Error);
	    END_IF;

	    // Energy save
	    #sR_TRIG_EnergySave(CLK := #iqUDT_Equipment.Report.EnergySave);                 // Energy save

	    IF #iqUDT_Equipment.Report.EnergySave OR #iqUDT_SystemControlCommand.ResetData  // Energy save
	    THEN
	        "FC_Statistics"(ix_Reset := #iqUDT_SystemControlCommand.ResetData,
	                        ix_Activate := #iqUDT_Equipment.Report.EnergySave,
	                        ix_RTrigActivate := #sR_TRIG_EnergySave.Q,
	                        iqUDT_Statistics := #iqUDT_Statistics.EnergySave);
	    END_IF;

	END_REGION

	REGION 11 – Reset the equipment states

	    #iqUDT_Equipment.Report.EnergySave := FALSE;           // Reset equipment report - energy save
	    #iqUDT_Equipment.Report.Error := FALSE;                // Reset equipment report - error
	    #iqUDT_Equipment.Report.Manual := FALSE;               // Reset equipment report - manual mode
	    #iqUDT_Equipment.Report.ManualRun := FALSE;            // Reset equipment report - run in manual mode
	    #iqUDT_Equipment.Report.AutoON := FALSE;               // Reset equipment report - automatic mode on
	    #iqUDT_Equipment.Report.Dieback := FALSE;              // Reset equipment report - dieback
	    #iqUDT_Equipment.Report.Halted := FALSE;               // Reset equipment report - halted
	    #iqUDT_Equipment.Report.SafetyStop := FALSE;           // Reset equipment report - safety stop
	    #iqUDT_Equipment.Report.Running := FALSE;              // Reset equipment report - started
	    #iqUDT_Equipment.Report.Stopped := FALSE;              // Reset equipment report - stopped
	    #iqUDT_Equipment.Report.Warning := FALSE;              // Reset equipment report - warning
	    #iqUDT_Equipment.Request.RestartRequired := FALSE;     // Reset equipment report - restart required

	END_REGION

	REGION 12 – Reset the HMI commands

	    #iqUDT_SystemControlCommand.Start := FALSE;             // Reset the HMI start command bit
	    #iqUDT_SystemControlCommand.Stop := FALSE;              // Reset the HMI stop command bit
	    #iqUDT_SystemControlCommand.ResetData := FALSE;         // Reset the HMI statistic reset bit
	    #iqUDT_SystemControlCommand.Reset := FALSE;             // Reset the HMI faults reset bit

	END_REGION
END_FUNCTION_BLOCK

FUNCTION_BLOCK "FB_VRCapacity"
{ S7_Optimized_Access := 'TRUE' }
VERSION : 0.1
// ATTRIBUTES
// AUTO_NUMBER = True
// BLOCK_NUMBER = 40
// END_ATTRIBUTES
   VAR_INPUT
      iUDT_CapacityConfiguration { ExternalAccessible := 'False'; ExternalVisible := 'False'; ExternalWritable := 'False'} : "UDT_CapacityConfiguration";   // Capacity configuration structure
      ix_PECFiltered { ExternalAccessible := 'False'; ExternalVisible := 'False'; ExternalWritable := 'False'} : Bool;   // TRUE when the end of section photoeye is not blocked
      ix_ResetData { ExternalAccessible := 'False'; ExternalVisible := 'False'; ExternalWritable := 'False'} : Bool;   // Reset data
   END_VAR

   VAR_OUTPUT
      qx_Error { ExternalAccessible := 'False'; ExternalVisible := 'False'; ExternalWritable := 'False'} : Bool;   // TRUE when collective block error occurred
      qx_Warning { ExternalAccessible := 'False'; ExternalVisible := 'False'; ExternalWritable := 'False'} : Bool;   // TRUE when collective block warning occurred
      qi_Capacity { ExternalAccessible := 'False'; ExternalVisible := 'False'; ExternalWritable := 'False'} : Int;   // Capacity value
      qa_CapacityBuffer { ExternalAccessible := 'False'; ExternalVisible := 'False'; ExternalWritable := 'False'} : Array[0..#Samples] of Int;   // Capacity buffer
      qa_PPHBuffer { ExternalAccessible := 'False'; ExternalVisible := 'False'; ExternalWritable := 'False'} : Array[0..#Samples] of Int;   // Parcel per hour buffer
   END_VAR

   VAR_IN_OUT
      iqUDT_ConveyorInterface : "UDT_ConveyorInterface";   // Conveyor interface
   END_VAR

   VAR
      sFB_Pulse { ExternalAccessible := 'False'; ExternalVisible := 'False'; ExternalWritable := 'False'; S7_SetPoint := 'False'} : "FB_Pulse";   // Function block to generate custom pulse signal.
      sR_TRIG_ParcelDetect {InstructionName := 'R_TRIG'; LibVersion := '1.0'; ExternalAccessible := 'False'; ExternalVisible := 'False'; ExternalWritable := 'False'; S7_SetPoint := 'False'} : R_TRIG;   // Parcel detect
      sa_Status { ExternalAccessible := 'False'; ExternalVisible := 'False'; ExternalWritable := 'False'} : Struct   // Status structure
         FifoError { ExternalAccessible := 'False'; ExternalVisible := 'False'; ExternalWritable := 'False'} : Bool;   //    FIFO block error
         FifoWarning { ExternalAccessible := 'False'; ExternalVisible := 'False'; ExternalWritable := 'False'} : Bool;   //    FIFO block warning
         ConfigurationError { ExternalAccessible := 'False'; ExternalVisible := 'False'; ExternalWritable := 'False'} : Bool;   //    Collective configuration error
      END_STRUCT;
      sr_CollectiveParcelLength { ExternalAccessible := 'False'; ExternalVisible := 'False'; ExternalWritable := 'False'} : Real;   // Colletive parcel length [mm]
      sr_ParcelCount { ExternalAccessible := 'False'; ExternalVisible := 'False'; ExternalWritable := 'False'} : Real;   // Parcel count
      sr_RecalculatedWindow { ExternalAccessible := 'False'; ExternalVisible := 'False'; ExternalWritable := 'False'} : Real;   // Window recalculated based on configured avg parcel length
      sr_ParcelPerHour { ExternalAccessible := 'False'; ExternalVisible := 'False'; ExternalWritable := 'False'} : Real;   // Parcel(s) per hour
      sr_AveragePackageLength { ExternalAccessible := 'False'; ExternalVisible := 'False'; ExternalWritable := 'False'} : Real;   // Average parcel length [mm]
      sr_AverageGap { ExternalAccessible := 'False'; ExternalVisible := 'False'; ExternalWritable := 'False'} : Real;   // Average gap size [mm]
      sr_AverageWindow { ExternalAccessible := 'False'; ExternalVisible := 'False'; ExternalWritable := 'False'} : Real;   // Average window size [mm]
      sudi_Interval { ExternalAccessible := 'False'; ExternalVisible := 'False'; ExternalWritable := 'False'} : UDInt;   // Interval [ms]
      si_Capacity { ExternalAccessible := 'False'; ExternalVisible := 'False'; ExternalWritable := 'False'} : Int;   // Capacity value for the configured package length
      si_ConveyorDistanceTraveled { ExternalAccessible := 'False'; ExternalVisible := 'False'; ExternalWritable := 'False'} : Int;   // Distance the conveyour travelled this interval
      sx_ParcelDetected { ExternalAccessible := 'False'; ExternalVisible := 'False'; ExternalWritable := 'False'} : Bool := FALSE;   // Parcel detected
      sx_SendData { ExternalAccessible := 'False'; ExternalVisible := 'False'; ExternalWritable := 'False'} : Bool;   // Send data signal
   END_VAR

   VAR CONSTANT
      Samples : ULInt := 120;
   END_VAR


BEGIN
	(*
	----------------------------------------------------------------------------------------

	Version history:
	Date        | Version   | Author        | Remark
	----------------------------------------------------------------------------------------
	21/01/2020  | 3.0       | A.Nowak       | Initial version
	14/02/2020  | 3.1       | A.Nowak       | Add sample amount and treshold to the configuration and reset data functionality
	13/03/2020  | 3.2       | M.Kurpiers    | Adapting reviews
	23/03/2020  | 3.3       | A. Nowak      | Change the values to the mm
	20/04/2022  | 3.4       | M.Roijen      | Remove MFC logging and added the shift of data
	06/08/2022  | 3.5       | M.Singh       | add Reset PPH Buffer and used avg Length from Config.
	15/05/2023  | 4.0       | F.Baten       | Lib 4.0
	                                          Removed Displacement memory, SampleAmount, fixed #sr_AveragePackageLength calculation.
	12/03/2024  | 4.1       | S. Nieswiec   | Small variable name changes according to current standard
	*)

	REGION 1 - Configuration check

	    // If the block is configured properly, convert interval to the ms and reset the error. Otherwise, set configuration error.
	    IF #iUDT_CapacityConfiguration.Interval > 0
	        AND #iUDT_CapacityConfiguration.AveragePackageLengthConfiguration > 0
	        AND #iUDT_CapacityConfiguration.Treshold >= 0
	    THEN
	        #sudi_Interval := #iUDT_CapacityConfiguration.Interval * 1000;
	        #sa_Status.ConfigurationError := FALSE;
	    ELSE
	        #sa_Status.ConfigurationError := TRUE;
	    END_IF;

	END_REGION

	REGION 2 - Reset data

	    // If there is reset data request, initialize sample amount and data buffer.
	    IF #ix_ResetData
	    THEN
	        FILL_BLK(IN := 0,
	                 COUNT := #Samples,
	                 OUT => #qa_CapacityBuffer[0]);
	        FILL_BLK(IN := 0,
	                 COUNT := #Samples,
	                 OUT => #qa_PPHBuffer[0]);
	    END_IF;

	END_REGION

	REGION 4 - PEC

	    #sx_ParcelDetected := NOT #ix_PECFiltered;

	END_REGION

	REGION 5 - Interval check

	    // Generate puls signal every interval.
	    #sFB_Pulse(iudi_PulseTime := #sudi_Interval,
	               qx_Pulse => #sx_SendData);

	END_REGION

	REGION 6 - Package length measurement and parcel count

	    // Parcel is detected.
	    IF #sx_ParcelDetected
	    THEN
	        // Add displacement to the collective parcel length.
	        #sr_CollectiveParcelLength += (ABS(#iqUDT_ConveyorInterface.Displacement)) * 10;
	    END_IF;

	    #sR_TRIG_ParcelDetect(CLK := #sx_ParcelDetected);
	    // Increment parcel count when package is detected.
	    IF #sR_TRIG_ParcelDetect.Q
	    THEN
	        #sr_ParcelCount += 1;
	    END_IF;

	    // Measure the distance traveled by conveyor
	    #si_ConveyorDistanceTraveled += (ABS(#iqUDT_ConveyorInterface.Displacement)) * 10;

	END_REGION

	REGION 7 - Capacity calculation and data send

	    // There is no configuration error and there are send data and enable signals.
	    IF NOT #sa_Status.ConfigurationError
	        AND #sx_SendData
	    THEN
	        // Parcel was detected.
	        IF #sr_ParcelCount <> 0
	            AND #sr_CollectiveParcelLength <> 0
	        THEN
	            // Calculate average values.
	            #sr_AveragePackageLength := #sr_CollectiveParcelLength / #sr_ParcelCount;
	            #sr_AverageWindow := #si_ConveyorDistanceTraveled / #sr_ParcelCount;
	            #sr_AverageGap := #sr_AverageWindow - #sr_AveragePackageLength;

	            // Windowsize calculated based on configured average parcel length
	            #sr_RecalculatedWindow := #sr_AverageGap + #iUDT_CapacityConfiguration.AveragePackageLengthConfiguration;

	            // Calculate parcel per hour value for the configured average parcel length.
	            #si_Capacity := DINT_TO_INT(TRUNC((#sr_ParcelPerHour * #sr_AverageWindow) / #sr_RecalculatedWindow));

	            // Calculate parcel per hour value using data from the interval.
	            #sr_ParcelPerHour := (#sr_ParcelCount / UDINT_TO_REAL(#iUDT_CapacityConfiguration.Interval)) * 3600;

	        ELSE
	            #si_Capacity := 0;
	        END_IF;

	        #qi_Capacity := #si_Capacity;

	        // Capacity value is greater than configured treshold.
	        IF #si_Capacity >= #iUDT_CapacityConfiguration.Treshold
	        THEN

	            MOVE_BLK(IN := #qa_CapacityBuffer[0],
	                     COUNT := #Samples,
	                     OUT => #qa_CapacityBuffer[1]);
	            #qa_CapacityBuffer[0] := #si_Capacity;

	            MOVE_BLK(IN := #qa_PPHBuffer[0],
	                     COUNT := #Samples,
	                     OUT => #qa_PPHBuffer[1]);
	            #qa_PPHBuffer[0] := REAL_TO_INT(#sr_ParcelPerHour);
	        END_IF;

	        // Initialize parcel count and collective parcel length.
	        #sr_ParcelCount := 0;
	        #sr_CollectiveParcelLength := 0;
	        #si_ConveyorDistanceTraveled := 0;
	    END_IF;

	END_REGION

	REGION 8 - Status

	    // Collective error.
	    #qx_Error :=
	    #sa_Status.ConfigurationError
	    OR #sa_Status.FifoError;

	    // Collective warning.
	    #qx_Warning := #sa_Status.FifoWarning;

	END_REGION
END_FUNCTION_BLOCK

